# B&R Automation Studio project TD52 (part 135)

#### de_excitCyclic.st
```iecst
(*******************************************************************************
de-excit	 deexcitation generator

This code is confidential and proprietary to the INNIO Company.
It may not be used in any form, or reproduced in any manner,
without the express written permission of the INNIO Company.
Copyright, INNIO Company, 2022

Customized modifications: -
------------------------

History:
-------
V2.12	24.04.2006	LH			copy of gcb
								adapted for de-exitation
		11.11.2006	LH			revised for final release after Para.bMSy test
V3.90.0	09.11.2012	lettenb.	new for modulare software project
		10.05.2013				rU_Gen_Nom --> rU_Gen_Nom[1]
V4.03.0 18.11.2015 	zengerer	BUGFIX Para.rU_Gen_Nom[1] <> 0
V4.07.0 01.02.2019	hohensinner	OUT_SY.bSel_DeExc New interfaces for CU Module (AB Energy like projects and so on), no functionality change in any module done! new INPUT interfaces are not connected! new OUTPUT interfaces are connected!
		17.05.2019	lettenb.	version
V4.09.0	28.11.2019	lettenb.	gen.deexcitation with closing gas valves(before with NOT bN_EngStart), to avoid undefined generator voltage values which may cause unwanted trips of protection relays(ThJ).
V4.10.0	24.11.2019	lettenb.	bMsg2354 added
V4.12.0	14.06.2022	lettenb.	tDemGenExcOff, tGenExcOff added, dead bb synch
		23.11.2022	lettenb.	bDeEx_Dem_x: bOMSS_Man, bOMSS_Aut removed(AA46/wasserer)
								ANW_ENTR: bGnlTrip1 -> bGnlTrip(same condition as for ton_gcb_dmnd_sy)(AA46/wasserer)
V4.13.0	17.08.2023	lettenb.	dead bb synch, bugfixes(BR21/wasserer,schwab,lettenb.)
		20.11.2023	Farre,		added IN_SY.bBypassMCB_SoftStart and soft energisation demand interfaces from CU needed for Microgrid (2023-168)
		29.11.2023	Goenczi,	demand de-exc. from HMI or BUS (e.g. Aggreko)

Instructions for use:
--------------------
Outstandings:
------------
*******************************************************************************)
PROGRAM _CYCLIC

	IF	Para.bSyActive AND Para.bGenDeexit_Enable	THEN

		(*----------------------------------------------------------------------------*)
		(* demand de-excitation *)
		bDeEx_Dem_Man	:=	bSyOMSS_Man
					AND	NOT	gcb.man_off
					AND	   ((gcb.man_on OR ANW_ENTR)
							OR (IN_SY.bOM_Bus				(*	either from HMI or BUS *)
								AND NOT IN_SY.bSetGCB2Open
								AND (IN_SY.bSetGCB2Close OR ANW_ENTR)));

		bDeEx_Dem_Aut	:=	bSyOMSS_Aut
					AND		IN_SY.bEng_Rdy_Aut_Exc;

		IF IN_SY.tDemGenExcOff.Di AND bP_Lo THEN (* dead bus synch *)
			ANW_ENTR	:= (bDeEx_Dem_Man OR bDeEx_Dem_Aut)
						OR (ANW_ENTR AND gcb.on);
		ELSE
			ANW_ENTR	:= (bDeEx_Dem_Man OR bDeEx_Dem_Aut OR IN_SY.bSoftEnergDem)
					AND	    bb_dead
					AND     gcb.eng_oper
					AND NOT gcb.on
					AND 	gcb.rel_trip
					AND 	(IN_SY.bBypassMCB_SoftStart OR (
							NOT		mcb.on
							AND 	mcb.remote
							AND 	mcb.racked_in))
					AND	NOT	bGnlTrip
					AND	NOT	bGen_DeExc_Err;
		END_IF;

		(*----------------------------------------------------------------------------*)
		(* generator de-excited (de-energized) *)
		bGen_DeExc_Rdy	:=	ANW_ENTR AND GEN_OSP;		(* feed-back generator without voltage    *)

		(*----------------------------------------------------------------------------*)
		(* de-excitation finished *)
		tof_T_ENTR(IN:=	ANW_ENTR, PT:= T#5s);

		OUT_SY.bGen_Exc_Off	:=	tof_T_ENTR.Q;

		(*----------------------------------------------------------------------------*)
		(* de-excitation failure *)
		ton_ST_ENTR(IN:= ANW_ENTR AND NOT GEN_OSP, PT:=	T#20s);
		tof_T_ST_ENTR(IN:= ton_ST_ENTR.Q, PT:= T#26s);

		bGen_DeExc_Err	:=	tof_T_ST_ENTR.Q;
		OUT_SY.bGen_DeExc_Rdy := bGen_DeExc_Rdy;
	ELSE
		ANW_ENTR		:= FALSE;
		OUT_SY.bGen_DeExc_Rdy := FALSE;
	END_IF;

	OUT_SY.bSel_DeExc	:=	ANW_ENTR;

		(*----------------------------------------------------------------------------*)
		(* Generator without voltage *)
		IF Para.rU_Gen_Nom[1] <> 0 THEN
			rU_Gen_Norm := IN_SY.tU_Avg[1].Ai / Para.rU_Gen_Nom[1];
		END_IF

		xGR_MIN_GEN_SPG(In:= rU_Gen_Norm, Gw:= Para.rU_Gen_DeEx_LimLo, Hy:= Para.rU_Gen_DeEx_LimLo/5);
		xTON_GEN_OSP(IN:= xGR_MIN_GEN_SPG.Q, PT:= T#1s);

		GEN_OSP := xTON_GEN_OSP.Q;
		OUT_SY.tGenExcOff.Do := GEN_OSP;

		bN_DeExc := IN_SY.rN_EngAct > (Para.rN_EngNom * 0.80);
		bDeEx_EngStop	:=	NOT bN_DeExc 	(* deexcitation at stopped engine, for unitrol reset *)
						AND NOT IN_SY.bGV_On
						AND NOT	IN_SY.bEng_Dem;

		(* Generator de-excitation *)
		bGenDeexitDem := (IN_SY.bMsg1036 OR IN_SY.bMsg1073 OR IN_SY.bMsg1132 OR IN_SY.bMsg1134 OR MM2VIS.bMsg2354 OR IN_SY.bMsg3319 OR ANW_ENTR OR bDeEx_EngStop)
				      AND(NOT IN_SY.tGCB_On.Di OR IN_SY.tDemGenExcOff.Di);
		OUT_SY.tGenDeexitDem.Do := bGenDeexitDem;

		(*----------------------------------------------------------------------------*)

END_PROGRAM
```

#### de_excit.var
```iecst
VAR
	bDeEx_Dem_Man : BOOL;
	bDeEx_Dem_Aut : BOOL;
	tof_T_ENTR : TOF;
	ton_ST_ENTR : TON;
	tof_T_ST_ENTR : TOF;
	xGR_MIN_GEN_SPG : GR_MINR;
	xTON_GEN_OSP : TON;
	bDeEx_EngStop : BOOL;
	bN_DeExc : BOOL;
END_VAR
```

### Program Logical/Synchronization/blackstart (IEC, version 4.13.0) - blackstart procedure

#### blackstartCyclic.st
```iecst
(*******************************************************************************
blackstart		blackout start

This code is confidential and proprietary to the INNIO Company.
It may not be used in any form, or reproduced in any manner,
without the express written permission of the INNIO Company.
Copyright, INNIO Company, 2022

Customized modifications: -
------------------------

History:
-------
V2.12	24.04.2006	LH			adapted for esy new
		02.10.2006	LH			modification of anti-detonation logic
		16.10.2006	LH			for execution load shedding:
								dmnd_load_shedd --> dmnd_black_start
		31.10.2006	LH			adaption of island release coming from Para.bMSy
		11.11.2006	LH			revised after Para.bMSy test
		20.11.2006	LH			revised for final release esy new
V2.20	27.04.2007	LH			update according to last changes mcb(s)
V2.20.1	08.08.2007	LH			termination of island power monitoring
V2.30	18.01.2008	LH			adapted for test-bench run
V3.99.0	04.03.2013	lettenb.	adapted for pilot engine 612, update anti detonation logic
		04.07.2013				IN_SY.tP_MnsImp_Act --> IN_SY.rP_MainsImport from MM_CU
V4.00.0 12.06.2014	lettenb.	test bTestBenchModeIsland
V4.03.0 18.11.2015  zengerer	BUGFIX NULLDIVISIONEN AND IN_SY.rP_Nom > 0
		11.04.2016	lettenb.	ton_dmnd_bs_over.Q -> dmnd_bs_over, bugfix
V4.12.0 29.06.2022	lettenb.	dead bb synch
V4.13.0 23.05.2023	Goenczi		code array view, interfaces from CU

Instructions for use:
--------------------

Outstandings:
------------
monitoring pmin in island operation ? (in v3.40 not active)
*******************************************************************************)
FUNCTION AND_Array
	memcpy(ADR(Arrayx),Adress,MIN(40,Size) + 1);
	AND_Array	:=	 TRUE;
	FOR i:= 0 TO MIN(40,Size) DO
		AND_Array	:=	AND_Array AND Arrayx[i];
	END_FOR
END_FUNCTION

FUNCTION OR_Array
	memcpy(ADR(Arrayx),Adress,MIN(40,Size) + 1);
	OR_Array	:=	 FALSE;
	FOR i:= 0 TO MIN(40,Size) DO
		OR_Array	:=	OR_Array OR Arrayx[i];
	END_FOR
END_FUNCTION

PROGRAM _CYCLIC

	IF	Para.bSyActive	THEN
		(*----------------------------------------------------------------------------*)
		(* general release island operation *)
		xTON_Sys_Run(IN:= IN_SY.tPB2MM.bSys_Run, PT:= T#10s);

		bIsl_mode[0]	:=	gcb.rel_island AND gcb.eng_oper AND gcb.other_gen_parallel AND	NOT	tof_mns_connection.Q;
		bIsl_mode[1]	:=	gcb.rel_island AND NOT OUT_SY.bSmoothDischarge;
		bIsl_mode[2]	:=	OUT_SY.bOnly_Island;

		bIsland_mode	:=	OR_Array(ADR(bIsl_mode),2);

		bRel_Isl[0]	:=	Para.bIslandOp_Enable OR Para.bOnlyIsland_Enable OR Para.bMSy OR Para.bMCB_Ctr_Cust	OR OUT_SY.bTestBenchModeIsland;
		bRel_Isl[1]	:=	IN_SY.tRel_I.Di;	(* release island extern (OUT_SY.bRel_Island)   *)
		bRel_Isl[2]	:=	xTON_Sys_Run.Q;
		bRel_Isl[3]	:=	bIsland_mode;
		bRel_Isl[4]	:=	IN_SY.bRel_I_Bus;	(*release island via Bus*)
		bRel_Isl[5]	:=	IN_SY.bCust_Rel_I;	(*custom release from CU*)

		bRelease_Island	:=	AND_Array(ADR(bRel_Isl),5);

		(* release island operation busbar: false = mains-cut-off with gcb *)
		bRel_Isl_BB[0]	:=	gcb.on AND bDem_Island AND NOT mcb.on;
		bRel_Isl_BB[1]	:=	gcb.on AND NOT sel_gcb_mains_cut_off AND NOT MM2VIS.bMsg3412;
		bRel_Isl_BB[2]	:=	other_gcb_on;
		bRel_Isl_BB[3]	:=	dmnd_black_start;
		bRel_Isl_BB[4]	:=	IN_SY.bCust_RelI_BB; 	(*new Aggreko release from CU*)
		bRel_Isl_BB[5]	:=	FALSE;

		bRelease_Isl_BB	:=	OR_Array(ADR(bRel_Isl_BB),5);

		bRel_VKE10[0]	:=	bRelease_Isl_BB;
		bRel_VKE10[1]	:=	bRelease_Island;
		bRel_VKE10[2]	:=	NOT	mcb.alm_psf OR	OUT_SY.bTestBenchModeIsland;
		bRel_VKE10[3]	:=	NOT	mcb.alm_opf;
		bRel_VKE10[4]	:=	NOT	any_gcb_opf_bb;

		bRelease_VKE10	:=	AND_Array(ADR(bRel_VKE10),4);

		(* demand island operation (INSEL) *)
		bDem_Isl[0]	:=	bRelease_VKE10;
		bDem_Isl[1]	:=	rel_i_adl OR NOT Para.bADL_Enable; (* release from anti-detonation logic *)

		bDem_Island	:=	AND_Array(ADR(bDem_Isl),1);

		(*----------------------------------------------------------------------------*)
		(* release black-out start *)
		rel_black_start	:= (Para.bBS_Enable OR Para.bOnlyIsland_Enable OR Para.bMSy	OR OUT_SY.bTestBenchModeIsland)
					AND		IN_SY.tRel_BS.Di;			(* release black-out extern (BL_OUT) *)

		(*----------------------------------------------------------------------------*)
		(* demand black-out start (BLOUT) *)
		black_status_bb := (all_gcb_off_bb OR IN_SY.tDemGenExcOff.Di)
					AND		mcb.off;

		(*----------------------------------------------------------------------------*)
		IF NOT Para.bMCB_ReSw2Mns_Enable THEN
			dmnd_black_start :=	bRelease_Island					(* BLOUT *)
						AND		rel_black_start
						AND	   (bSyOMSS_Man OR	NOT	Para.bBS_OnlyMan)
						AND	   (bOMSS_Man   OR	NOT	Para.bBS_OnlyMan)
						AND(NOT bMainsReturn					    OR black_status_bb)
						AND	   (mcb.off     OR  NOT MM2VIS.bMsg3412 OR black_status_bb)
						AND   	mcb.remote
						AND(NOT	mcb.alarm   OR	    OUT_SY.bTestBenchModeIsland)
						AND NOT any_gcb_alarm_bb
						AND NOT	dmnd_bs_over;

		ELSIF Para.bMCB_ReSw2Mns_Enable THEN
			dmnd_black_start :=	bRelease_Island					(* BLOUT *)
						AND		rel_black_start
						AND	   (bSyOMSS_Man OR	NOT	Para.bBS_OnlyMan)
						AND	   (bOMSS_Man   OR	NOT	Para.bBS_OnlyMan)
						AND	NOT bMainsReturn
						AND	   (mcb.off     OR  NOT MM2VIS.bMsg3412)
						AND   	mcb.remote
						AND(NOT	mcb.alarm   OR	    OUT_SY.bTestBenchModeIsland)
						AND NOT any_gcb_alarm_bb
						AND NOT	dmnd_bs_over;
		END_IF;

		(*----------------------------------------------------------------------------*)
		(* black-out start procedure finished *)
		dmnd_bs_over	:= (dmnd_black_start OR	dmnd_bs_over)
					AND		gcb.eng_oper
					AND		gcb.on;

		(*----------------------------------------------------------------------------*)
		(* demand load shedding *)
		dmnd_load_shedd	:=	black_status_bb
					AND		bRelease_Island
					AND		rel_black_start
					AND		dmnd_black_start;

		(* load shedding ok *)
		ton_ls_ok(IN:= dmnd_load_shedd AND IN_SY.tRel_LS.Di, PT:= T#5s);

		rel_load_shedd	:=	ton_ls_ok.Q;		(* load shedding is done (LAST_AB) *)

		(******************************************************************************)
		(* anti detonation logic *)
		(*----------------------------------------------------------------------------*)
		tof_mns_connection(IN:= mcb.on, PT:= T#5s);	(* mains connected to busbar	 *)
		ton_gcb_on        (IN:=	gcb.on, PT:= T#5s);	(* generator connected to busbar *)

		(*----------------------------------------------------------------------------*)
		IN_SY.rP_Nom;						(* engine nominal generator power [kW] *)
		IN_SY.rP_Act_Norm_Filt;				(* engine actual  generator power [kW] *)

		rPchange_max	:=	40.0;			(* maximum allowed loss of gen. power *)
		rPgen_min		:=	15.0;			(* minimum required island power      *)

		(*----------------------------------------------------------------------------*)
		(* generator power supplied to busbar *)
		IF gcb.on THEN	rP_Gen_Act_Norm := IN_SY.rP_Act_Norm_Filt;
		ELSE			rP_Gen_Act_Norm := 0.0;
		END_IF;

		(* mains power to busbar in % Pnom engine *)
		IF mcb.on AND IN_SY.rP_Nom > 0  THEN	rP_Mns_Act_Norm := IN_SY.rP_MainsImport / IN_SY.rP_Nom;
		ELSE			rP_Mns_Act_Norm := 0.0;
		END_IF;

		(* consumer load on busbar *)
		rP_Csm_Act_Norm := rP_Gen_Act_Norm + rP_Mns_Act_Norm;

		(*----------------------------------------------------------------------------*)
		(* release for island operation *)
		IF (Para.bMSy AND mcb.on AND bRelease_VKE10) OR NOT mcb.on THEN
			rel_i_adl		:=	TRUE;
		ELSIF NOT VKE41 AND mcb.on	THEN
			rel_i_adl		:=	TRUE;					(* cond. to change into island are ok *)
		ELSE
			rel_i_adl		:=	FALSE;					(* change into island is not allowed  *)
		END_IF;

		(*----------------------------------------------------------------------------*)
		(* monitoring change of generator power in case of opening mcb *)
		VKE40			:=	VKE41						(* maintained lock command            *)
					AND	NOT	gcb.on
					AND		gcb.eng_run;

		VKE41			:=	VKE40						(* --> lock module after opening xcb  *)
					OR	   (rPchange > rPchange_max);	(* because of too much loss of power  *)

		(* --> no load expected because:  *)
		bPcalc		:=		mcb.on								(* - no connection to mains          *)
					AND		bRelease_VKE10						(* - no island operation selected    *)
					AND		(IN_SY.rP_MainsImport <> -999999.0)	(* - no mains power signal, value if signal not connected = -999999 from MM_CU *)
					AND		other_gcb_off;						(* - Pcsm calculation  not possible	*)

		IF	bPcalc	THEN
			rP_I_Act_Norm_Expected := rP_Csm_Act_Norm;	(* gen.load will be consumer load   *)
		ELSE
			rP_I_Act_Norm_Expected := 0;				(* no load expected at opening xcb    *)
		END_IF;

		(* change of gen. power at opening xcb = generator power supplied to busbar - expect.load in case of opening mcb*)
		rPchange	:=	IN_SY.rP_Act_Norm_Filt - rP_I_Act_Norm_Expected;

		(*----------------------------------------------------------------------------*)

	END_IF;

END_PROGRAM
```

#### blackstartInit.st
```iecst
PROGRAM _INIT
	(* init program *)

	rPel_csm_old	:=	10000.0;

END_PROGRAM
```

#### blackstart.fun
```iecst
(********************************************************************
 * COPYRIGHT -- INNIO Company
 ********************************************************************
 * Package: blackstart
 * File: blackstart.fun
 * Author: 212426533
 * Created: November 29, 2023
 *******************************************************************)

FUNCTION AND_Array : BOOL
	VAR_INPUT
		Adress : UDINT;
		Size : USINT;
	END_VAR
	VAR
		i : USINT;
		Arrayx : ARRAY[0..40] OF BOOL;
	END_VAR
END_FUNCTION

FUNCTION OR_Array : BOOL
	VAR_INPUT
		Adress : UDINT;
		Size : USINT;
	END_VAR
	VAR
		i : USINT;
		Arrayx : ARRAY[0..40] OF BOOL;
	END_VAR
END_FUNCTION
```

#### blackstart.var
```iecst
VAR
	rPchange : REAL;
	rPchange_max : REAL;
	rPel_csm_old : REAL;
	rPgen_min : REAL;
	rP_Gen_Act_Norm : REAL;
	rP_Mns_Act_Norm : REAL;
	rP_Csm_Act_Norm : REAL := 0.0;
	tof_mns_connection : TOF;
	ton_gcb_on : TON;
	ton_ls_ok : TON;
	black_status_bb : BOOL;
	xTON_Sys_Run : TON;
	dmnd_bs_over : BOOL;
	bRelease_VKE10 : BOOL; (* release island operation busbar: false = mains-cut-off with gcb *)
	VKE40 : BOOL;
	VKE41 : BOOL;
	bPcalc : BOOL;
	dmnd_load_shedd : BOOL; (*Demand load shed*)
	rP_I_Act_Norm_Expected : REAL;
	bIsl_mode : ARRAY[0..2] OF BOOL := [3(0)];
	bIsland_mode : BOOL := 0;
	bRel_Isl : ARRAY[0..5] OF BOOL := [6(0)];
	bRel_Isl_BB : ARRAY[0..5] OF BOOL := [6(0)]; (* release island operation busbar condition OR array: false = mains-cut-off with gcb *)
	bRelease_Isl_BB : BOOL := 0; (* release island operation busbar part1 *)
	bDem_Isl : ARRAY[0..1] OF BOOL := [2(0)]; (* demand island operation (INSEL) condition array*)
	bRel_VKE10 : ARRAY[0..4] OF BOOL := [5(0)]; (* release island operation busbar condition AND array: false = mains-cut-off with gcb *)
END_VAR
```

### Program Logical/Synchronization/sy_out (IEC, version 4.13.0) - out signals handling

#### sy_outCyclic.st
```iecst
(*******************************************************************************
sy_out		control outputs

This code is confidential and proprietary to the INNIO Company.
It may not be used in any form, or reproduced in any manner,
without the express written permission of the INNIO Company.
Copyright, INNIO Company, 2022

Customized modifications: -
------------------------

History:
-------
V2.12	24.04.2006	LH			gcb1 imported from MSY
								gcb1 --> sy_out
								adapted for esy new
		31.10.2006	LH			insert release gcb from Para.bMSy
		11.11.2006	LH			revised after Para.bMSy test
		20.11.2006	LH			revised for final release esy new
V2.20	07.02.2007	LH			new: lock command for customer mcb
		19.02.2007	LH			adapted for X20-system
								advanced software documentation
		04.04.2007	LH			correction of OUT_SY.bRel_IslandAfMITime in case of mcb controlled by customer
V2.201	22.05.2007	TW			change MMU variables to array (ex task: DO)
V2.30	16.01.2008	LH			building OUT_SY.bRel_IslandAfMITime to prevent engine shutdown
								during waiting time for island demand
		18.01.2008	LH			adapted for test-bench run
V2.30	22.02.2008	LH			change output gcb opening failure (ex task: DO)
		26.02.2008	LH			connect gcb position sig. fail. to engine control
		05.03.2008	LH			change gcb position sig. fail. to engine control
								to undelayed tripping
		28.03.2008	LH			connect gcb closing failure to engine control
V2.34.0	19.12.2008	lettenb.	OUT_SY.bRelEngOpFromSY: gcb.mdl removed
V2.60.0	13.08.2009	lettenb.	gcb_opf_delay for opening mcb with delay added (ex task: DO)
V2.60.0	08.10.2009	lettenb.	ton_dmnd_synchline added (delay for activating synch.device
 								after switching on the voltage signals to the synch.device.
								MMUsynch needs some time until frequence measuring is ok)
V3.20.0	01.07.2010	lettenb.	BR9_B added
		13.01.2011	lettenb.	Para.bEngOpAfterMIF_Enable added
V3.20.0	04.11.2010	lettenb.	bSyncSlipMode[2], bMMU2syMCB added for synchr.mcb with MMU2 (ex task: DO)
V3.30.0 02.02.2012	lettenb.	OUT_SY.bEng_Dem_EPS_Sy: Para.bIslandOp_Enable	added(to avoid message 'demand emerg.operation'
								in case of mains break down and no island operation is selected)
V3.90.0	13.11.2012	lettenb.	parts from pb17_en included
V3.99.0 26.02.2013	lettenb.	task DO included, iEngNr added
V3.99.1	25.03.2013	Denk		bRelSyFromCU changed to bRelSy_Customized
		27.06.2013	lettenb.	bRelEng4OnlyI_Op: brackets added, bugfix
V4.00.0 11.06.2014	lettenb.	bRelEng4I_Op: logic, ton_BLO_AES.PT case iEngNr, bugfix
		16.06.2014	lettenb.	OUT_SY.bRelEngOpFromSy: IN_SY.tMCB_Rel_Sync_SOn.Do ERDF lockout added (grid)
V4.04.0 31.10.2016				ton_esl.IN: ... AND FALSE) (* FALSE=econ_lock; added, acc.a_V3.59, wasserer/rosenheim)
        05.12.2016				OUT_SY.tRdy_MSy.Do,OUT_SY.tEng_Run_Sy.Do,OUT_SY.tEng_Dem.Do always active for GSY
		01.10.2020	lettenb.	OUT_SY.bMCB_DemSy, mcb controlled by customer, bugfix(heim, Referenzanlage AB85), bu
V4.10.0 15.12.2020	lettenb.	BR6 release island after MIF: bRel_IslandAfMITime in case of Para.bP_LoadReject_Active AND IN_SY.bType6_Update_Rel
V4.12.0 24.11.2020	lettenb.	WaitingTime_CloseGCB2DeadBB_too_long issue#911
								xTOF_RelEng4I_Op added, avoid loss of RelEng4I_Op for 1 cycle at OMSS change to OFF in island, issue#957
V4.13.0	17.08.2023	lettenb.	dead bb synch, bugfixes(BR21/wasserer,schwab,lettenb.)
		19.07.2023	Goenczi		Added Para.bSel_Customer to bRelEng4I_Op to bypass Dem_Island for Aggreko
								bEng_Dem_EPS_Sy condition from CU module added

Instructions FOR use:
--------------------
						variante:	ESy		+Msy	+CCB	noSy	GSy		AB_Sy
	immer	A_USP
			DO_ENG_D
			DO_PUL_MNS_OK
			DO_GCB_REL
			DO_GCB_RSP
			DO_GCB_OPF
			DO_GCB_CON
			DO_GCB_COF
			DO_GCB_RT

	msy		DO_GCB_ESL
			DO_GCB_EDC
			DO_RDY_MSY
			DO_ENG_RUN		OUT_SY.tEng_Run.Do;

	mcb		DO_MCB_RSP
			DO_MCB_DVS
			DO_MCB_RT
			DO_MCB_CON
			DO_MCB_COF

	AB		A_SYANW
			A_RSYANW

	indon.	DO_DMND_LS

Outstandings:
------------
define variations by parameter-settings
*******************************************************************************)
PROGRAM _CYCLIC

	IF	Para.bSyActive	THEN
		(*----------------------------------------------------------------------------*)
		(* demand synchline *)			(* OUT_SY.bDSyLine *)
		ton_dmnd_synchline(IN:= (gcb.dmnd_sy OR mcb.dmnd_sy) AND NOT pulse_sy_line, PT:= T#2s);

		dmnd_synchline := ton_dmnd_synchline.Q;

		(*----------------------------------------------------------------------------*)
		(* ESy demand lock all other cb's for closing gcb to dead busbar *)		(* BLO_AES) *)
		ton_BLO_AES.IN	:= (ton_gcb_dmnd_sy.IN	OR ton_gcb_dmnd_sy.Q)
					AND(    bb_dead OR(IN_SY.tDemGenExcOff.Di AND NOT bb_alive))(* dead busbar (OUT_SY.bBB_dead) *)
					AND(NOT	MM2VIS.bMsg1216	OR	OUT_SY.bTestBenchModeIsland)	(* no busbar voltage sensor failure *)
					AND(NOT any_gcb_on_bb   OR  IN_SY.tDemGenExcOff.Di)			(* all gcb open - busbar *)
					AND	NOT any_gcb_psf_bb										(* no other gcb with position failure *)
					AND NOT any_gcb_opf_bb										(* no other gcb with opening failure *)
					AND NOT mcb.on												(* all mcb open *)
					AND(NOT mcb.alm_psf		OR	OUT_SY.bTestBenchModeIsland)	(* no mains cb with position failure *)
					AND		IN_SY.tPB2MM.bSys_Run;								(* CPU is alive *)

		IF Para.bMSy THEN
			ton_BLO_AES.PT	:=	T#1s;		(* gcb close2deadBB interlock is done MSy *)
		ELSE
			CASE iEngNr OF
			1:	ton_BLO_AES.PT	:=	T#1s;	(* engine 1 *)
			2:	ton_BLO_AES.PT	:=	T#2s;
			3:	ton_BLO_AES.PT	:=	T#3s;
			4:	ton_BLO_AES.PT	:=	T#4s;
			5:	ton_BLO_AES.PT	:=	T#5s;
			6:	ton_BLO_AES.PT	:=	T#6s;
			7:	ton_BLO_AES.PT	:=	T#7s;
			8:	ton_BLO_AES.PT	:=	T#8s;
			9:	ton_BLO_AES.PT	:=	T#9s;
			10:	ton_BLO_AES.PT	:=	T#10s;
			11:	ton_BLO_AES.PT	:=	T#11s;
			12:	ton_BLO_AES.PT	:=	T#12s;
			13:	ton_BLO_AES.PT	:=	T#13s;
			14:	ton_BLO_AES.PT	:=	T#14s;
			15:	ton_BLO_AES.PT	:=	T#15s;
			16:	ton_BLO_AES.PT	:=	T#16s;
			ELSE
				ton_BLO_AES.PT	:=	T#17s;
			END_CASE;
		END_IF;
		ton_BLO_AES();

		gcb.edc		:=	ton_BLO_AES.Q									(* demand closing gcb to dead busbar *)
					OR	mcb_man_on2dead_bb								(* manual closing mcb1 to dead busbar *)
					OR	mcb_aut_on2dead_bb;								(* automatic closing mcb1 to dead busbar *)

		(* ESY demand lock customer mcb while running island operation *)
		BLOCK_NS		:=	ton_BLO_AES.Q								(* demand closing gcb to dead busbar *)
					OR(			BLOCK_NS
						AND		any_gcb_on_bb							(* lock customer mcb will last until *)
						AND	NOT	mcb.dmnd_sy);							(* resynchronizing is initiated *)

		(* release closing cb to dead busbar to MSY/external unit (AES_FRG) *)
		ton_esl.IN		:= (bb_dead AND NOT	ton_gcb_dmnd_sy.IN AND IN_SY.tPB2MM.bSys_Run AND NOT gcb.release AND FALSE) (* FALSE= ex.econ_lock;	interlock cb's only with 1 signal ? *)
					OR	   (any_gcb_edc_bb	                   AND IN_SY.tPB2MM.bSys_Run AND NOT gcb.release)			(* demand closing ext. cb to dead busbar (ANF_BLO) *)
					OR	   (gcb.mdl                            AND IN_SY.tPB2MM.bSys_Run AND NOT gcb.release);			(* demand lock from MSy *)
		ton_esl(PT:= T#1s);												(* engine (gcb) status locked -> release gcb (FG_GS) *)

		gcb.esl		:=	ton_esl.Q;										(* release closing ext. cb to dead busbar (AES_FRG) *)

		(*----------------------------------------------------------------------------*)
		(* demand emergency operation (OUT_SY.bEng_Dem_EPS_Sy) *)
		OUT_SY.bEng_Dem_EPS_Sy	:= ((Para.bIslandOp_Enable OR Para.bOnlyIsland_Enable OR Para.bMSy OR Para.bMCB_Ctr_Cust)
							AND(NOT	mains.ok OR	NOT	mcb.on)
							AND IN_SY.bCust_Dem_EPS_Sy);

		(*----------------------------------------------------------------------------*)
		(* release engine operation from ESY (OUT_SY.bRelEngOpFromSY) *)
		bRelEng4NP_Op	:= (mains.ok OR gcb.eng_oper)					(* release for parallel operation *) (* mehrfachverwendung *)
					AND		mcb.on										(* mcb closed (NS(1)_EIN) *)
					AND		bMainsReturn								(* mains return (OUT_SY.bMainsReturn) *)
					AND	NOT	MM2VIS.bMsg3412;							(* mains monitoring device failure *)

		(*----------------------------------------------------------------------------*)
		(* hold release engine for island op. after mi-filter time *)
		xTOF_Rel_IslandAfMITime(IN:= mains.ok, PT:= T#60s);

		IF 			NOT	gcb.eng_oper									(* no engine operation (IN_SY.tEng_Run.Do) *)
				OR	NOT	Para.bMIF_Enable
				OR		Para.bBS_OnlyMan
				OR	NOT	Para.bEngOpAfterMIF_Enable
				OR	   (xEngType.Type6 AND (NOT Para.bP_LoadReject_Active OR NOT IN_SY.bType6_Update_Rel))
				OR		xEngType.Type9
		THEN
			xTOF_Rel_IslandAfMITime(IN:= FALSE, PT:= T#0s); 			(* reset bridging *)
		END_IF;

		OUT_SY.bRel_IslandAfMITime	:=	xTOF_Rel_IslandAfMITime.Q;		(* prevention of engine shutdown (M_BLOCK) *)
		(*----------------------------------------------------------------------------*)

		(* hold release engine for island op. for reswitch to mains *)
		xTOF_Rel_Island4Resw2Mns(IN:= gcb.on, PT:= T#60s);

		IF		NOT	gcb.eng_oper										(* no engine operation (IN_SY.tEng_Run.Do) *)
			OR	NOT	Para.bMCB_ReSw2Mns_Enable
			OR		Para.bBS_OnlyMan
			OR	   (xEngType.Type6 AND (NOT Para.bP_LoadReject_Active OR NOT IN_SY.bType6_Update_Rel))
			OR		xEngType.Type9
		THEN
			xTOF_Rel_Island4Resw2Mns(IN:= FALSE, PT:= T#0s);			(* reset bridging *)
		END_IF;

		bRel_Island4Resw2Mns := xTOF_Rel_Island4Resw2Mns.Q;

		(*----------------------------------------------------------------------------*)
		xTOF_RelEng4I_Op(IN	:= (Para.bIslandOp_Enable OR Para.bMSy OR Para.bMCB_Ctr_Cust OR OUT_SY.bTestBenchModeIsland)
						AND	   (rel_i_adl OR NOT Para.bADL_Enable)
						AND	   (OUT_SY.bRel_IslandAfMITime OR bRel_Island4Resw2Mns OR bDem_Island OR gcb.rel_trip OR Para.iSel_Customer = 2), PT:= T#200ms);
		bRelEng4I_Op	:= xTOF_RelEng4I_Op.Q;

		bRelEng4OnlyI_Op:=	OUT_SY.bOnly_Island
					AND		mcb.off
					AND	NOT	mcb.on
					AND	  ((OUT_SY.bRelEngOpFromSy AND(gcb.eng_oper OR gcb.eng_demanded)) OR NOT gcb.eng_run);

		bRelEng4Op		:=	mcb.remote
					AND		mcb.racked_in
					AND		gcb.racked_in
					AND  (((bRelEng4NP_Op OR bRelEng4I_Op) AND NOT OUT_SY.bOnly_Island) OR bRelEng4OnlyI_Op);	(* release for island/parallel operation *)

		OUT_SY.bRelEngOpFromSy := 	IN_SY.tLineCB_On.Di
								AND IN_SY.bRelSy_Customized				(* from MM_CU *)
								AND bRelEng4Op
								AND IN_SY.tMCB_Rel_Sync_SOn.Do;			(* ERDF lockout *)
	ELSE

		OUT_SY.bRelEngOpFromSy := 	IN_SY.tLineCB_On.Di
								AND IN_SY.bRelSy_Customized 			(* from MM_CU *)
								AND IN_SY.tRelEngOpFromGSy.Di
								AND IN_SY.tMCB_Rel_Sync_SOn.Do;			(* ERDF lockout *)
	END_IF;

	(*-----------------------------------------------------------------------------*)
	(* diagnostics *)
	bRelEng4NP_Op;				(* release engine for net parallel *)
	bRelEng4I_Op;				(* release engine for island(emergency op.)*)
	bRelEng4OnlyI_Op;			(* release engine for only island *)
	OUT_SY.bRelEngOpFromSy;		(* release engine for operation from sy *)
	(*-----------------------------------------------------------------------------*)

	(*-----------------------------------------------------------------------------*)
	(* switch standard-inputs esy to required inputs engine control *)
		OUT_SY.bSynchDem		:=		IN_SY.tGCB_DSY.Di;				(* demand synchline *)

		(* general -------------------------------------------------------------------*)
		OUT_SY.tRdy_MSy.Do		:=		IN_SY.bEng_Rdy_Aut_Exc;			(* engine ready    for MSY/GSY *)
		OUT_SY.tEng_Run_Sy.Do	:=		bN_EngStart;					(* engine rotating for MSY/GSY *)
		OUT_SY.tEng_Dem.Do		:=		IN_SY.bEng_RPSDem;				(* engine demanded for MSY/GSY *)
		OUT_SY.tOMSS_Man.Do		:=		bOMSS_Man;						(* oper.mode man.  for     GSY *)
		OUT_SY.tOMSS_Aut.Do		:=		bOMSS_Aut;						(* oper.mode aut.  for     GSY *)

	IF	Para.bSyActive	THEN
		OUT_SY.tDemandBB.Do		:=		gcb.dmnd_sy;					(* demand busbar *)

		OUT_SY.tGCB_ESL.Do		:=		gcb.esl;						(* ESY status gcb locked *)
		OUT_SY.tGCB_EDC.Do		:=		gcb.edc;						(* ESY demand lock all other cb's connected to dead busbar *)
		OUT_SY.tLock_C_MCB.Do	:=		BLOCK_NS;						(* demand lock customer mcb while running island operation *)
		OUT_SY.tGCB_OpF.Do		:=		gcb_opf_delay;					(* alarm gcb opening failure *)

		(* generator circuit breaker -------------------------------------------------*)
		OUT_SY.tGCB_Rel.Do		:=		gcb.release;					(* release closing gcb *)
		OUT_SY.tGCB_RSP.Do		:=		gcb.rel_sy_puls;				(* release sy pulse gcb *)
		OUT_SY.tGCB_COn.Do		:=		gcb.command_on;					(* command gcb on *) (* Do = true  = command ON  *)
		OUT_SY.tGCB_COf.Do		:=	NOT gcb.command_off;				(* command gcb off *)(* Do = false = command OFF, closed circuit principle *)
		OUT_SY.tGCB_RT.Do		:=		gcb.rel_trip;					(* release trip gcb *)
		OUT_SY.tGCB_DVS.Do		:=		gcb.dmnd_sy;					(* demand synchronization gcb - select voltage *)

		(* mains circuit breaker -----------------------------------------------------*)
		OUT_SY.tMCB_RSP.Do		:=	NOT Para.bMSy AND mcb.rel_sy_puls;	(* release sy pulse mcb1 *)
		OUT_SY.tMCB_COn.Do		:=	NOT Para.bMSy AND mcb.command_on;	(* command mcb1 on *)
		OUT_SY.tMCB_COf.Do		:=	NOT Para.bMSy AND mcb.command_off;	(* command mcb1 off *)
		OUT_SY.tMCB_RT.Do		:=	NOT Para.bMSy AND mcb.rel_trip;		(* release trip mcb1 *)
		OUT_SY.tMCB_DVS.Do		:=	NOT Para.bMSy AND mcb.dmnd_sy;		(* demand synchronization mcb1 - select voltage *)

		(* switch standard-outputs esy to standard-inputs engine control -------------*)
		OUT_SY.bMsg1217			:=		gcb.alm_psf;					(* alarm gcb position signal failure *)
		OUT_SY.bMsg1218			:=		gcb.alm_opf;					(* alarm gcb opening failure *)
		OUT_SY.bMsg1219			:=		gcb.alm_cf;						(* alarm gcb closing failure *)
		bGCB_GnlWarning			:=		gcb.alarm;						(* gcb general warning *)
		OUT_SY.bMsg1209			:=		mcb.alm_psf;					(* alarm mcb position signal failure *)
		bMCB_GnlWarning			:=		mcb.alarm;						(* mcb general warning *)

		OUT_SY.bGCB_DemSy		:=		gcb.dmnd_sy;					(* demand synchronization gcb for main loop display *)
		OUT_SY.bMCB_DemSy		:=		mcb.dmnd_sy AND Para.bMCB_Enable;(* demand synchronization mcb for main loop display *)
		OUT_SY.bDSyLine			:=		dmnd_synchline;					(* ESY demand synchline for synchronizing gcb *)
		OUT_SY.bMnsOk			:=		IN_SY.tMnsOk.Di;				(* mains ok       for W1175 *)
		OUT_SY.bMainsReturn		:=		bMainsReturn;					(* mains return   for W1175 and block engine *)
		OUT_SY.bBB_dead			:=		bb_dead;						(* busbar dead for main loop display and B2139/B3265 *)
		OUT_SY.bRel_Island		:=		bRelease_Island;				(* release island for W1175 and block engine *)
		BLOUT					:=		dmnd_black_start;				(* demand black-out start for demand load shedding *)
		OUT_SY.bOtherGenParallel:=		OUT_SY.bOtherGenParallel;		(* other engine parallel for demand emergency op. *)

		(* switch standard-outputs esy new to standard-inputs MMU/Sync ---------------*)
		OUT_SY.bSyncSlipMode[1] :=	   (OUT_SY.bMCB_DemSy	AND NOT Para.bMCB_SyMMD2)	(* synchronization with slip mode *)
									OR (OUT_SY.bGCB_DemSy	AND	NOT	bb_dead);
		OUT_SY.bSyncSlipMode[2] :=  	OUT_SY.bMCB_DemSy	AND 	Para.bMCB_SyMMD2;	(* synchronization with slip mode *)

		(*----------------------------------------------------------------------------*)
		(* synchronizing device on *)			(* SYG_EIN *)
		OUT_SY.bGen_SyD_Dem 	:= (gcb.dmnd_sy OR mcb.dmnd_sy) AND	bb_alive;

		(* release synchronizing pulse *)		(* FG_SYIMP *)
		ton_dmnd_sy_device(IN:= OUT_SY.bGen_SyD_Dem, PT:= T#2s);
		rel_sy_puls				:=	ton_dmnd_sy_device.Q;

		(*----------------------------------------------------------------------------*)
	END_IF;

END_PROGRAM
```

#### sy_out.var
```iecst
VAR
	ton_BLO_AES : TON;
	ton_esl : TON;
	xTOF_Rel_IslandAfMITime : TOF;
	xTOF_Rel_Island4Resw2Mns : TOF;
	ton_dmnd_synchline : TON;
	bRel_Island4Resw2Mns : BOOL;
	bRelEng4NP_Op : BOOL; (* release engine for net parallel operation*)
	bRelEng4I_Op : BOOL; (* release engine for island operation*)
	bRelEng4OnlyI_Op : BOOL; (* release engine for only island operation*)
	bRelEng4Op : BOOL;
	ton_dmnd_sy_device	:TON;
	xTOF_RelEng4I_Op : TOF;
END_VAR
```

### Program Logical/Synchronization/vis_SY (IEC, version 4.13.0) - visualization

#### vis_SYCyclic.st
```iecst
(*******************************************************************************
vis_SY			visualization

This code is confidential and proprietary to the INNIO Company.
It may not be used in any form, or reproduced in any manner,
without the express written permission of the INNIO Company.
Copyright, INNIO Company, 2022

Customized modifications: -
------------------------

History:
-------
V3.90.0	17.10.2012	lettenb.	new
V3.99.0	04.03.2013	lettenb.	new version
V4.07.0	11.10.2018	lettenb.	DI/DO dataitems for diagnosis added
 		25.04.2019	lettenb.	dataitem changed IN_SY.tGCB_DVM.Di, bugfix
		01.10.2020	lettenb.	MM2VIS.bDSyMCB, mcb controlled by customer, bugfix(heim, Referenzanlage AB85), bu
V4.12.0	14.09.2022	lettenb.	MM2VIS.bDemGenExcOff, MM2VIS.bGenExcOff added, dead bb synch
V4.13.0	29.11.2023	Goenczi		bGCB_OGP_Bus other genset paralell bit via bus

Instructions for use:
--------------------
Outstandings:
------------
*******************************************************************************)
PROGRAM _CYCLIC

	MM2VIS.bMnsOk			:=		OUT_SY.bMnsOk;		(* mains ok *)
	MM2VIS.bNotMainsReturn	:=	NOT	bMainsReturn;		(* not mains return *)

	MM2VIS.bGCB_On			:=		IN_SY.tGCB_On.Di;	(* gcb closed for report time measuring *)
	MM2VIS.bGCB_GnlWarning	:=		bGCB_GnlWarning;	(* gcb general failure *)
	MM2VIS.bDSyGCB			:=		gcb.dmnd_sy;		(* gcb demand synchronization *)

	MM2VIS.bMCB_On			:=		OUT_SY.bMCB_On;		(* mcb closed for report time measuring *)
	MM2VIS.bMCB_GnlWarning	:=		bMCB_GnlWarning;	(* mcb general failure *)
	MM2VIS.bDSyMCB			:=		mcb.dmnd_sy AND Para.bMCB_Enable;	(* mcb demand synchronization *)

	MM2VIS.bEngDemIsland 	:=		IN_SY.tEngDemIsland.Di;	(* DI engine demand for island operation *)
	MM2VIS.bOnly_Island		:=		IN_SY.tOnly_Island.Di;	(* DI only island operation *)
	MM2VIS.bGCB_MDL			:=		IN_SY.tGCB_MDL.Di;		(* DI generator circuit breaker master demand lock (for closing other GCB to dead BB) *)
	MM2VIS.bGCB_MRC			:=		IN_SY.tGCB_MRC.Di;		(* DI generator circuit breaker master release close (to dead busbar) *)
	MM2VIS.bGCB_AGO			:=		IN_SY.tGCB_AGO.Di;		(* DI all other generator circuit breaker off *)
	MM2VIS.bGCB_RI			:=		IN_SY.tGCB_RI.Di;		(* DI generator circuit breaker reelase island *)
	MM2VIS.bGCB_OGP			:=		IN_SY.tGCB_OGP.Di OR IN_SY.bGCB_OGP_Bus;		(* DI generator circuit breaker other generator parallel *)
	MM2VIS.bGCB_DVM			:=		IN_SY.tGCB_DVM.Di;		(* DI voltage matching for synchronization *)
	MM2VIS.bGCB_DSY			:=		IN_SY.tGCB_DSY.Di;		(* DI generator circuit breaker demand synchronization (synchline) *)
//	MM2VIS.bF_N_DI_Inc		:=		IN_OP.tF_N_DI_Inc.Di;	(* DI synch.increase speed *)
//	MM2VIS.bF_N_DI_Dec		:=		IN_OP.tF_N_DI_Dec.Di;	(* DI synch.decrease speed *)
//	MM2VIS.bU_Gen_Inc		:=		IN_GC.tU_Gen_Inc.Di;	(* DI voltage adjustment external (increasing)*)
//	MM2VIS.bU_Gen_Dec		:=		IN_GC.tU_Gen_Dec.Di;	(* DI voltage adjustment external (decreasing)*)

	MM2VIS.bRdy_MSy			:=		OUT_SY.tRdy_MSy.Do;		(* DO engine ready    for MSY/GSY *)
	MM2VIS.bEng_Run_Sy		:=		OUT_SY.tEng_Run_Sy.Do;	(* DO engine rotating for MSY/GSY *)
	MM2VIS.bEng_Dem			:=		OUT_SY.tEng_Dem.Do;		(* DO engine demanded for MSY/GSY *)
	MM2VIS.bGCB_OpF			:=		OUT_SY.tGCB_OpF.Do;		(* DO alarm gcb opening failure *)
	MM2VIS.bGCB_EDC			:=		OUT_SY.tGCB_EDC.Do;		(* DO ESY demand lock all other cb's connected to dead busbar *)
	MM2VIS.bGCB_ESL			:=		OUT_SY.tGCB_ESL.Do;		(* DO ESY status gcb locked *)

//	MM2VIS.bImp_OpHour  	:= 		OUT_OP.tImp_OpHour.Do;	(* DO Impulse for operation hour counter *)
//	MM2VIS.bEng_Rdy_Rem 	:= 		OUT_OP.tEng_Rdy_Rem.Do;	(* DO Ready for Remote Operation *)
//	MM2VIS.bEng_Run 		:=		OUT_OP.tEng_Run.Do;		(* DO Engine in operation*)

	MM2VIS.bDemGenExcOff	:=		IN_SY.tDemGenExcOff.Di;	(* DI demand generator excitation off*)
	MM2VIS.bGenExcOff		:=		OUT_SY.tGenExcOff.Do;	(* DO generator excitation off*)

END_PROGRAM
```

### Program Logical/Synchronization/PermSY (IEC, version 4.10.0) - + PermanentMemory

- PermSYCyclic.st (not readable text: treated as protected, skipped)

- PermSYInit.st (not readable text: treated as protected, skipped)

#### PermSY.var
```iecst
VAR
	pm_Error : UINT;
	write_once : BOOL;
	pm_len : UDINT;
	ModulName : STRING[35];
	DatObjInfo_01 : DatObjInfo;
	pm_id : UDINT;
	pm_p : UDINT;
	bCreateDataObj : BOOL;
	perm_par_vers : UINT;
	DatObjRead_01 : DatObjRead;
	DatObjDelete_PermMem : DatObjDelete;
	DatObjCreate_01 : DatObjCreate;
	DatObjWrite_01 : DatObjWrite;
	ulChecksumOld : UDINT;
	ulPMPointer : UDINT;
	ulChkValue : UDINT;
	TON_WritePMEM : TON;
	ulChecksum : UDINT;
	bWriteDataObj : BOOL;
	TON_WarnDelay : TON;
	TON_BlockMinFileAge : TON; (*waiting time without file write after successful performed write*)
	bBlock_MinFileAge : BOOL := FALSE; (*pause the perm file write after each sucessful write*)
	iPM_WriteCnt : UDINT; (* *) (*old VarName: usPMWriteCnt*)
END_VAR
VAR CONSTANT
	ERR_NOERROR : UINT := 0;
END_VAR
VAR
	pmm : Perm_SY_Struct;
END_VAR
```

### Program Logical/Synchronization/ParSY (IEC, version 4.06.0) - + parameter handling

- perm_par.st (not readable text: treated as protected, skipped)

#### perm_par.var
```iecst
VAR
	tParaIntern : ParaHandler_typ; (*Connector type to perm_par*)
	tMM2ParaBase_ReadBack : MM2ParaBase_type; (*INTERNAL! V4.06 new readback structure for information from previous tasks*)
	bWriteDataObj : BOOL; (* TRUE=write data object module *)
	bDataObjLenErr : BOOL; (*Error occured in permem: data module size missmatch*)
	bCreateDataObj : BOOL; (* TRUE=create new data object *)
	bWriteOnce : BOOL; (* write permanent memory once *)
	DatObjCreate_01 : DatObjCreate; (* data object create *)
	DatObjInfoBak_02 : DatObjInfo; (* data object info *)
	DatObjDelete_01 : DatObjDelete; (* data object delete *)
	DatObjRead_01 : DatObjRead; (* data object read *)
	DatObjRead_02 : DatObjRead; (* manual initiated data object read *)
	DatObjWrite_01 : DatObjWrite; (* data object write *)
	DatObjDelete_02 : DatObjDelete; (* data object delete *)
	DatObjDelete_11 : DatObjDelete; (*Delete Backup File*)
	DatObjInfo_01 : DatObjInfo; (* data object info *)
	DatObjInfo_02 : DatObjInfo; (* data object info *)
	szModuleName : STRING[35]; (* module name of object *)
	szModuleNameBackup : STRING[35]; (* module name of posiibly created backup object *)
	DatObjCopy_01 : DatObjCopy;
	bCopyDataObj : BOOL;
	TON_WarnDelay : TON;
	TON_WritePMEM : TON; (* delay write permanent memory *)
	ulPMPointer : UDINT; (* adress of actual checksum value *)
	ulChecksum : UDINT; (* parameter checksum value *)
	pm_len : UDINT; (* permanent value lenght *)
	ulChecksumOld : UDINT; (* last vlaue of parameter checksum *)
	ulChkValue : UDINT; (* actual value of parameter pointer *)
	pm_id : UDINT; (* permanent value identifier *)
	pm_p : UDINT; (* permanent value pointer *)
	DatObjInfo_META : DatObjInfo;
	DatObjRead_META : DatObjRead;
	szMetaDataRaw : STRING[2000];
	szMetaData : ARRAY[0..4] OF STRING[35];
	szMetaDataVis : ARRAY[0..3] OF STRING[35];
	ssIndex : INT;
	ssCount : INT;
	ucMetaDataRaw : ARRAY[0..2000] OF USINT;
	ssCount2 : INT;
	szMetaDataFile : STRING[10];
	szText1 : STRING[20];
	pv_adr_IN_XX_tPB2MM : UDINT;
	pv_lng : UDINT;
	pv_lng_IN_XX_tPB2MM : UDINT;
	pv_lng_OUT_XX_tPB2MM : UDINT;
	szText2 : STRING[20];
	pv_adr_OUT_XX_tXX2PB : UDINT;
END_VAR
VAR CONSTANT
	ERR_NOERROR : UINT := 0;
END_VAR
VAR
	usPMWriteCnt : UINT;
	pm_Error : UDINT; (* permanent value error *) (* Deleted: pm : ParaMem_typ; permanent memory tags mathias, 22.8.11*)
	fun_Error : UDINT := 0; (*state > 0 = function error*)
	xLocalParaCheck : ParaCheckFUB; (*local function instance to check parameter values*)
	TON_ParaSetupOk : TON;
	bParaCheckSystemOk : BOOL;
	iDebug_ParaOkChecked : UDINT;
	bRestoreBackupDataObj : BOOL := FALSE;
	bRestoreDataObjContent : BOOL := FALSE;
	pm_id_backup : UDINT;
	pm_p_Backup : UDINT;
	DatObjCopy_02 : DatObjCopy;
	bDeleteBackupDataObj : BOOL := FALSE; (*Command to delete backup data module file on purpose*)
	bDebugPara : ARRAY[0..5] OF BOOL;
	ssIndex2 : INT;
	ssIndex3 : INT;
	ssIndex4 : INT;
	ssIndexVis : INT;
	szText : STRING[40];
	pv_adr_Para : UDINT;
	szParaSnippet : ARRAY[0..5] OF STRING[150];
	szParaIndex : STRING[10];
	slValue : DINT;
	iModuleDLD_ResetCount : INT;
	bDownloadDetected : BOOL;
	bFlagParaStructCopyWorking : BOOL; (*true, if cyclic para copying is active, 1 false cycle at every copy *)
	bStoreInitParaInDataObj : BOOL := FALSE;
	bTestflag : BOOL;
	bReadOutMETA_Once : BOOL;
	tParaCheck_iPvAdress : ARRAY[0..5] OF UDINT;
	tParaCheck_iPvLengt : ARRAY[0..5] OF UDINT;
	tParaCheck_rPvValue : ARRAY[0..5] OF REAL;
	tParaCheck_rRangeMIN : ARRAY[0..5] OF REAL;
	tParaCheck_rRangeMAX : ARRAY[0..5] OF REAL;
	tParaCheck_szPvName : ARRAY[0..5] OF STRING[35];
	ssFormatDetected : INT;
	szMetaDataPart : STRING[150];
	szFullTaskName : STRING[35];
	szFullMetaModuleName : STRING[35];
	debugLen : INT;
	debugSize : INT := 0;
	strcat_adr1 : UDINT;
	strcat_adr2 : UDINT;
	ssIndexTN : INT;
	bAlternate : BOOL;
	n : INT;
	iAlternateChecksum : DINT;
	iAlternateChecksumOld : DINT;
	ulDebugChkValue : ARRAY[0..999] OF UDINT;
	Adr1 : UDINT;
	Adr2 : UDINT;
	usPMWriteCntStepsize : UINT := 1; (*different step sizes to help debug*)
	usPMWriteCntXOR : UINT;
	usPMWriteCntAltSum : UINT;
	ulAdrPM : UDINT;
	usChkValuePM : USINT;
	ulAdrPara : UDINT;
	ulPara_len : UDINT;
	usChkValuePara : USINT;
	iDebugCountPMDifferences : DINT := 0;
	bEngineRunDetected : BOOL; (*detection status bit autocommand 100 /101  for engine run state*)
	ucMetaDataDebugInfoLine : ARRAY[0..24] OF STRING[80];
	ssIndexMand : INT := 0;
	szMetaDataMand : STRING[35];
	iMyErrorInfo_Autoreset : DINT; (*internal autoreset counter*)
	ssIndex_Version : INT; (*internal*)
	ssIndex_BU : INT; (*internal*)
	ssIndex_BU2 : INT; (*internal*)
END_VAR
```

### Program Logical/Synchronization/LV_GCB (IEC) - LV GCB communication

#### LV_GCB_Cyclic.st - Cyclic
```iecst
(*******************************************************************************
AGGR: Modbus RTU connection to LV GCB  (cyclic)

This code is confidential and proprietary to the INNIO Company.
It may not be used in any form, or reproduced in any manner, without the express
written permission of the INNIO Company.
Copyright, INNIO Company, 2023

Customized modifications: -
------------------------

History:
-------
V4.13	14-11-2023	Hohensinner	created

Instructions for use:
--------------------
Caution!
- X20CS1030_xxx_xx_GCB should not be in "cyclic stream" mode, instead it should be set to "stream".
- Also the modules name must be ending with "_GCB" to be found in the init part.

Outstandings:
------------
*******************************************************************************)

PROGRAM _CYCLIC

	(** 1: waiting for parasetup okay *)
	xTON_ParaSetup_Ok(IN:= TRUE AND NOT bError_Conf, PT:= tiParaSetup_Ok);
	IF NOT xTON_ParaSetup_Ok.Q OR bDeactivate_Task OR DiagCpuIsSimulated() THEN RETURN; END_IF

	(** 2: running the modbus master *)
	xTON_Rel_MBMaster(IN:= xTON_ParaSetup_Ok.Q, PT:=tiRel_MBMaster);
	xMBDO_Master[0].bEnable	:=	xTON_Rel_MBMaster.Q;
	xMBDO_Master[0]();

	(** 3: State Machine of LV GCB connection *)
	CASE eState_GCB OF
		_GCB_INIT:
			eState_GCB := _GCB_TRY_ABB;
		_GCB_TRY_ABB:
			(* Init *)
			IF bInit THEN
				tSlave[0].tLine[0].tIF.bExec	:=	TRUE;	//make first contact
			END_IF
			(* Wait *)
			xWAIT(IN:=1);
			(* Exit *)
			IF xWAIT.Q THEN
				IF 	NOT tSlave[0].tLine[0].tIF.bExec AND tSlave[0].tLine[0].tIF.iStatus = 0 THEN
					eState_GCB := _GCB_IDLE;
					MM2VIS.tGCB[1].iType	:= 1;
				ELSIF tSlave[0].tLine[0].tIF.bExec AND tSlave[0].tLine[0].tIF.iStatus <> ERR_FUB_BUSY THEN
					eState_GCB := _GCB_TRY_SE;
					tSlave[0].tLine[0].tIF.bExec	:=	FALSE;	//end first contact
				END_IF
			END_IF
		_GCB_TRY_SE:
			(* Init *)
			IF bInit THEN
				tSlave[1].tLine[0].tIF.bExec	:=	TRUE;	//make first contact
			END_IF
			(* Wait *)
			xWAIT(IN:=1);
			(* Exit *)
			IF xWAIT.Q THEN
				IF 	NOT tSlave[1].tLine[0].tIF.bExec AND tSlave[1].tLine[0].tIF.iStatus = 0 THEN
					eState_GCB := _GCB_IDLE;
					MM2VIS.tGCB[1].iType	:= 2;
				ELSIF tSlave[1].tLine[0].tIF.bExec AND tSlave[1].tLine[0].tIF.iStatus <> ERR_FUB_BUSY THEN
					eState_GCB := _GCB_WAIT;
					tSlave[1].tLine[0].tIF.bExec	:=	FALSE;	//end first contact
				END_IF
			END_IF
		_GCB_WAIT:
			(* Wait *)
			xWAIT(IN:=100);
			(* Exit *)
			IF xWAIT.Q THEN
				eState_GCB := _GCB_TRY_ABB;
			END_IF
		_GCB_CALC:
			FOR i:=0 TO 60 DO
				rFactors := 0.4 + UINT_TO_REAL(i) * 0.01;
				IF VIS2MM.tGCB[1].rI_GenNom * 1.1 <= rFactors * MM2VIS.tGCB[1].rI_Nom THEN
					EXIT;
				END_IF
			END_FOR
			VIS2MM.tGCB[1].rI1	:=	MM2VIS.tGCB[1].rI_Nom * rFactors;
			IF bSE THEN
				VIS2MM.tGCB[1].rt1	:=	1;
			ELSIF bABB THEN
				VIS2MM.tGCB[1].rt1	:=	3;
			END_IF
			VIS2MM.tGCB[1].rI2	:=	MM2VIS.tGCB[1].rI_Nom * 2;
			VIS2MM.tGCB[1].rt2	:=	0.3;
			VIS2MM.tGCB[1].rI3	:=	MM2VIS.tGCB[1].rI_Nom * 10;
			eState_GCB := _GCB_IDLE;
		_ABB_LOAD:
			(* Init *)
			IF bInit THEN
				VIS2MM.tGCB[1].rI_GenNom := Para.rI_GenNom[1];
				tSlave[0].tLine[6].tIF.bExec	:=	TRUE;
				tSlave[0].tLine[7].tIF.bExec	:=	TRUE;
				tSlave[0].tLine[8].tIF.bExec	:=	TRUE;
				tSlave[0].tLine[12].tIF.bExec	:=	TRUE;
			END_IF
			(* Wait *)
			xWAIT(IN:=1);
			MM2VIS.tGCB[1].rLoad	:=	BOOL_TO_REAL(NOT tSlave[0].tLine[6].tIF.bExec)/4
									+	BOOL_TO_REAL(NOT tSlave[0].tLine[7].tIF.bExec)/4
									+	BOOL_TO_REAL(NOT tSlave[0].tLine[8].tIF.bExec)/4
									+	BOOL_TO_REAL(NOT tSlave[0].tLine[12].tIF.bExec)/4;
			(* Exit *)
			IF NOT tSlave[0].tLine[6].tIF.bExec AND NOT tSlave[0].tLine[7].tIF.bExec AND
				NOT tSlave[0].tLine[8].tIF.bExec AND NOT tSlave[0].tLine[12].tIF.bExec AND xWAIT.Q THEN
				MM2VIS.tGCB[1].rI_Nom			:=	UINT_TO_REAL(tSlave[0].tLine[12].tIF.iData[0]);
				VIS2MM.tGCB[1].rI1				:=	MM2VIS.tGCB[1].rI_Nom * UINT_TO_REAL(tSlave[0].tLine[6].tIF.iData[1])/1000;
				VIS2MM.tGCB[1].rt1				:=	UINT_TO_REAL(tSlave[0].tLine[6].tIF.iData[2])/100;
				VIS2MM.tGCB[1].rI2				:=	MM2VIS.tGCB[1].rI_Nom * UINT_TO_REAL(tSlave[0].tLine[7].tIF.iData[1])/100;
				VIS2MM.tGCB[1].rt2				:=	UINT_TO_REAL(tSlave[0].tLine[7].tIF.iData[2])/100;
				VIS2MM.tGCB[1].rI3				:=	MM2VIS.tGCB[1].rI_Nom * UINT_TO_REAL(tSlave[0].tLine[8].tIF.iData[1])/100;
				eState_GCB := _ABB_READ;
			END_IF
		_ABB_READ:
			(* Init *)
			IF bInit THEN
				tSlave[0].tLine[0].tIF.bExec	:=	TRUE;
				tSlave[0].tLine[2].tIF.bExec	:=	TRUE;
				tSlave[0].tLine[3].tIF.bExec	:=	TRUE;
				tSlave[0].tLine[4].tIF.bExec	:=	TRUE;
				tSlave[0].tLine[11].tIF.bExec	:=	TRUE;
				tSlave[0].tLine[12].tIF.bExec	:=	TRUE;
			END_IF
			(* Wait *)
			xWAIT(IN:=1);
			(* Exit *)
			IF 	NOT tSlave[0].tLine[0].tIF.bExec AND
				NOT tSlave[0].tLine[2].tIF.bExec AND
				NOT tSlave[0].tLine[3].tIF.bExec AND
				NOT tSlave[0].tLine[4].tIF.bExec AND
				NOT tSlave[0].tLine[11].tIF.bExec AND
				NOT tSlave[0].tLine[12].tIF.bExec AND xWAIT.Q THEN
				MM2VIS.tGCB[1].rWear			:=	UINT_TO_REAL(tSlave[0].tLine[0].tIF.iData[0])/65000;
				MM2VIS.tGCB[1].iNumOp			:=	UINT_TO_DINT(tSlave[0].tLine[0].tIF.iData[1]);
				MM2VIS.tGCB[1].iNumPT			:=	UINT_TO_DINT(tSlave[0].tLine[0].tIF.iData[3]);
				MM2VIS.tGCB[1].rI_Act_L1		:=	(UINT_TO_REAL(tSlave[0].tLine[2].tIF.iData[0])+UINT_TO_REAL(tSlave[0].tLine[2].tIF.iData[1])*65536)/10;
				MM2VIS.tGCB[1].rI_Act_L2		:=	(UINT_TO_REAL(tSlave[0].tLine[2].tIF.iData[2])+UINT_TO_REAL(tSlave[0].tLine[2].tIF.iData[3])*65536)/10;
				MM2VIS.tGCB[1].rI_Act_L3		:=	(UINT_TO_REAL(tSlave[0].tLine[2].tIF.iData[4])+UINT_TO_REAL(tSlave[0].tLine[2].tIF.iData[5])*65536)/10;
				MM2VIS.tGCB[1].rU_Act			:=	UINT_TO_REAL(tSlave[0].tLine[3].tIF.iData[0])/10/3
												+	UINT_TO_REAL(tSlave[0].tLine[3].tIF.iData[1])/10/3
												+	UINT_TO_REAL(tSlave[0].tLine[3].tIF.iData[2])/10/3;
				MM2VIS.tGCB[1].rU_Nom			:=	UINT_TO_REAL(tSlave[0].tLine[4].tIF.iData[0]);
				MM2VIS.tGCB[1].bClosed			:=	tSlave[0].tLine[11].tIF.iData[0].0;
				MM2VIS.tGCB[1].bRacked			:=	tSlave[0].tLine[11].tIF.iData[0].1;
				MM2VIS.tGCB[1].bFail			:=	tSlave[0].tLine[11].tIF.iData[0].13
												OR	tSlave[0].tLine[11].tIF.iData[0].7
												OR NOT tSlave[0].tLine[11].tIF.iData[0].8
												OR	tSlave[0].tLine[11].tIF.iData[0].10
												OR	tSlave[0].tLine[11].tIF.iData[0].5;
				MM2VIS.tGCB[1].rI_Nom			:=	UINT_TO_REAL(tSlave[0].tLine[12].tIF.iData[0]);
				bABB_Remote						:= tSlave[0].tLine[11].tIF.iData[0].8;
				eState_GCB := _GCB_IDLE;
			END_IF
		_ABB_SAVE_OPEN:
			(* Init *)
			IF bInit THEN
				tSlave[0].tLine[13].tIF				:=	tIF_ABB_Open;
				MM2VIS.tGCB[1].rSave				:=	0.33;
			END_IF
			(* Wait *)
			xWAIT(IN:=1);
			(* Exit *)
			IF NOT tSlave[0].tLine[13].tIF.bExec AND xWAIT.Q THEN
				eState_GCB := _ABB_SAVE_DATA;
			END_IF
		_ABB_SAVE_DATA:
			(* Init *)
			IF bInit THEN																												//LOW	HIGH	STEP
				tSlave[0].tLine[14].tIF.iData[0]	:=	LIMIT(REAL_TO_UINT(VIS2MM.tGCB[1].rI1/MM2VIS.tGCB[1].rI_Nom*1000),400,1000);	//400	1000	1
				tSlave[0].tLine[14].tIF.iData[1]	:=	LIMIT(REAL_TO_UINT(VIS2MM.tGCB[1].rt1),3,144)*100;								//300	14400	100
				tSlave[0].tLine[9].tIF.iData[0]		:=	LIMIT(REAL_TO_UINT(VIS2MM.tGCB[1].rI2/MM2VIS.tGCB[1].rI_Nom*10),6,100)*10;		//60	1000	10
				tSlave[0].tLine[9].tIF.iData[1]		:=	LIMIT(REAL_TO_UINT(VIS2MM.tGCB[1].rt2*100),5,80);								//5		80		1
				tSlave[0].tLine[10].tIF.iData[0]	:=	LIMIT(REAL_TO_UINT(VIS2MM.tGCB[1].rI3/MM2VIS.tGCB[1].rI_Nom*10),15,150)*10;		//150	1500	10
				tSlave[0].tLine[14].tIF.bExec		:=	TRUE;
				tSlave[0].tLine[9].tIF.bExec		:=	TRUE;
				tSlave[0].tLine[10].tIF.bExec		:=	TRUE;
				MM2VIS.tGCB[1].rSave				:=	0.66;
			END_IF
			(* Wait *)
			xWAIT(IN:=1);
			(* Exit *)
			IF NOT tSlave[0].tLine[14].tIF.bExec AND NOT tSlave[0].tLine[9].tIF.bExec AND NOT tSlave[0].tLine[10].tIF.bExec AND xWAIT.Q THEN
				eState_GCB := _ABB_SAVE_CLOSE;
			END_IF
		_ABB_SAVE_CLOSE:
			(* Init *)
			IF bInit THEN
				tSlave[0].tLine[13].tIF		:=	tIF_ABB_Close;
			END_IF
			(* Wait *)
			xWAIT(IN:=1);
			(* Exit *)
			IF NOT tSlave[0].tLine[13].tIF.bExec AND xWAIT.Q THEN
				eState_GCB := _ABB_LOAD;
				MM2VIS.tGCB[1].rSave				:=	1.00;
			END_IF
		_SE_LOAD:
			(* Init Load *)
			IF bInit THEN
				VIS2MM.tGCB[1].rI_GenNom := Para.rI_GenNom[1];
				tSlave[1].tLine[4].tIF.bExec	:=	TRUE;	//to load I_Nom
				tSlave[1].tLine[6].tIF.bExec	:=	TRUE;
				tSlave[1].tLine[7].tIF.bExec	:=	TRUE;
				tSlave[1].tLine[8].tIF.bExec	:=	TRUE;
			END_IF
			(* Wait Load *)
			xWAIT(IN:=1);
			MM2VIS.tGCB[1].rLoad	:=	BOOL_TO_REAL(NOT tSlave[1].tLine[4].tIF.bExec)/4
									+	BOOL_TO_REAL(NOT tSlave[1].tLine[6].tIF.bExec)/4
									+	BOOL_TO_REAL(NOT tSlave[1].tLine[7].tIF.bExec)/4
									+	BOOL_TO_REAL(NOT tSlave[1].tLine[8].tIF.bExec)/4;
			(* Exit Load *)
			IF NOT tSlave[1].tLine[4].tIF.bExec AND NOT tSlave[1].tLine[6].tIF.bExec AND NOT tSlave[1].tLine[7].tIF.bExec AND NOT tSlave[1].tLine[8].tIF.bExec AND xWAIT.Q THEN
				MM2VIS.tGCB[1].rI_Nom	:=	UINT_TWO_REAL(tSlave[1].tLine[4].tIF.iData[2],tSlave[1].tLine[4].tIF.iData[3]);
				VIS2MM.tGCB[1].rI1	:=	UINT_TWO_REAL(tSlave[1].tLine[6].tIF.iData[0],tSlave[1].tLine[6].tIF.iData[1]);
				VIS2MM.tGCB[1].rt1	:=	UINT_TWO_REAL(tSlave[1].tLine[6].tIF.iData[2],tSlave[1].tLine[6].tIF.iData[3]);
				rFactor_Isd			:=	UINT_TWO_REAL(tSlave[1].tLine[7].tIF.iData[0],tSlave[1].tLine[7].tIF.iData[1]);
				VIS2MM.tGCB[1].rI2	:=	rFactor_Isd*VIS2MM.tGCB[1].rI1;
				VIS2MM.tGCB[1].rt2	:=	UINT_TWO_REAL(tSlave[1].tLine[7].tIF.iData[2],tSlave[1].tLine[7].tIF.iData[3]);
				rFactor_Ii			:=	UINT_TWO_REAL(tSlave[1].tLine[8].tIF.iData[1],tSlave[1].tLine[8].tIF.iData[2]);
				VIS2MM.tGCB[1].rI3	:=	rFactor_Ii*MM2VIS.tGCB[1].rI_Nom;
				eState_GCB := _SE_READ;
			END_IF
		_SE_READ:
			(* Init Read *)
			IF bInit THEN
				tSlave[1].tLine[0].tIF.bExec	:=	TRUE;
				tSlave[1].tLine[1].tIF.bExec	:=	TRUE;
				tSlave[1].tLine[2].tIF.bExec	:=	TRUE;
				tSlave[1].tLine[3].tIF.bExec	:=	TRUE;
				tSlave[1].tLine[4].tIF.bExec	:=	TRUE;
				tSlave[1].tLine[5].tIF.bExec	:=	TRUE;
//				tSlave[1].tLine[9].tIF.bExec	:=	TRUE;		//falls SE racked in / out IO interface besitzt aktivieren
			END_IF
			(* Wait Read *)
			xWAIT(IN:=1);
			(* Exit Read *)
			IF 	NOT tSlave[1].tLine[0].tIF.bExec AND
				NOT tSlave[1].tLine[1].tIF.bExec AND
				NOT tSlave[1].tLine[2].tIF.bExec AND
				NOT tSlave[1].tLine[3].tIF.bExec AND
				NOT tSlave[1].tLine[4].tIF.bExec AND
				NOT tSlave[1].tLine[5].tIF.bExec AND
				NOT tSlave[1].tLine[9].tIF.bExec AND xWAIT.Q THEN
				MM2VIS.tGCB[1].iNumOp			:=	UDINT_TO_DINT(UINT_TWO_UDINT(tSlave[1].tLine[0].tIF.iData[0],tSlave[1].tLine[0].tIF.iData[1]));
				MM2VIS.tGCB[1].iNumPT			:=	UDINT_TO_DINT(UINT_TWO_UDINT(tSlave[1].tLine[0].tIF.iData[2],tSlave[1].tLine[0].tIF.iData[3]));
				MM2VIS.tGCB[1].rI_Act_L1		:=	UINT_TWO_REAL(tSlave[1].tLine[2].tIF.iData[0],tSlave[1].tLine[2].tIF.iData[1]);
				MM2VIS.tGCB[1].rI_Act_L2		:=	UINT_TWO_REAL(tSlave[1].tLine[2].tIF.iData[2],tSlave[1].tLine[2].tIF.iData[3]);
				MM2VIS.tGCB[1].rI_Act_L3		:=	UINT_TWO_REAL(tSlave[1].tLine[2].tIF.iData[4],tSlave[1].tLine[2].tIF.iData[5]);
				MM2VIS.tGCB[1].rU_Act			:=	UINT_TWO_REAL(tSlave[1].tLine[3].tIF.iData[0],tSlave[1].tLine[3].tIF.iData[1]);
				MM2VIS.tGCB[1].rU_Nom			:=	UINT_TWO_REAL(tSlave[1].tLine[4].tIF.iData[0],tSlave[1].tLine[4].tIF.iData[1]);
				MM2VIS.tGCB[1].rI_Nom			:=	UINT_TWO_REAL(tSlave[1].tLine[4].tIF.iData[2],tSlave[1].tLine[4].tIF.iData[3]);
				MM2VIS.tGCB[1].rWear			:=	UINT_TWO_REAL(tSlave[1].tLine[5].tIF.iData[0],tSlave[1].tLine[5].tIF.iData[1]);
				MM2VIS.tGCB[1].bClosed			:=	tSlave[1].tLine[1].tIF.iData[1].0;
				MM2VIS.tGCB[1].bRacked			:=	tSlave[1].tLine[9].tIF.iData[0].9;
				eState_GCB := _GCB_IDLE;
			END_IF
		_SE_SAVE_CHECK:												 //Check if no session is open
			(* Init Check *)
			IF bInit THEN
				tSlave[1].tLine[11].tIF.bExec		:=	TRUE;
				MM2VIS.tGCB[1].rSave				:=	0.1;
			END_IF
			(* Wait Check *)
			xWAIT(IN:=1);
			(* Exit Check *)
			IF NOT tSlave[1].tLine[11].tIF.bExec AND xWAIT.Q THEN
				IF (tSlave[1].tLine[11].tIF.iData[3] <> 0 OR tSlave[1].tLine[11].tIF.iData[4] <> 0) AND tSlave[1].tLine[11].tIF.iData[0]<>1933 THEN
					iSessionKey0 := tSlave[1].tLine[11].tIF.iData[3];
					iSessionKey1 := tSlave[1].tLine[11].tIF.iData[4];
					eState_GCB := _SE_SAVE_CLOSE_OLD;
				ELSE
					eState_GCB := _SE_SAVE_OPEN;
				END_IF
			END_IF
		_SE_SAVE_CLOSE_OLD:								//close old session
			(* Init Close *)
			IF bInit THEN
				tSlave[1].tLine[10].tIF 			:=	tIF_Session_Close;
				tSlave[1].tLine[10].tIF.iData[6]	:=	iSessionKey0;
				tSlave[1].tLine[10].tIF.iData[7]	:=	iSessionKey1;
				MM2VIS.tGCB[1].rSave				:=	0.2;
			END_IF
			(* Wait Close *)
			xWAIT(IN:=1);
			(* Exit Close *)
			IF NOT tSlave[1].tLine[10].tIF.bExec AND xWAIT.Q THEN
				eState_GCB := _SE_SAVE_OPEN;
			END_IF
		_SE_SAVE_OPEN:										//open new session
			(* Init Open *)
			IF bInit THEN
				tSlave[1].tLine[10].tIF 			:=	tIF_Session_Open;
				MM2VIS.tGCB[1].rSave				:=	0.3;
			END_IF
			(* Wait Open *)
			xWAIT(IN:=1);
			(* Exit Open *)
			IF NOT tSlave[1].tLine[10].tIF.bExec AND xWAIT.Q THEN
				eState_GCB := _SE_SAVE_ID;
			END_IF
		_SE_SAVE_ID:										//ask for new session ID
			(* Init ID *)
			IF bInit THEN
				tSlave[1].tLine[11].tIF.bExec		:=	TRUE;
				MM2VIS.tGCB[1].rSave				:=	0.4;
			END_IF
			(* Wait ID *)
			xWAIT(IN:=1);
			(* Exit ID *)
			IF NOT tSlave[1].tLine[11].tIF.bExec THEN
				IF tSlave[1].tLine[11].tIF.iData[1] = 0 AND tSlave[1].tLine[11].tIF.iData[2] = 4 AND xWAIT.Q THEN
					iSessionKey0 := tSlave[1].tLine[11].tIF.iData[3];
					iSessionKey1 := tSlave[1].tLine[11].tIF.iData[4];
					eState_GCB := _SE_SAVE_DATA1;
				ELSE
					iSessionKey0 := tSlave[1].tLine[11].tIF.iData[3];
					iSessionKey1 := tSlave[1].tLine[11].tIF.iData[4];
					eState_GCB := _SE_SAVE_CLOSE_OLD;
				END_IF
			END_IF
		_SE_SAVE_DATA1:											//change Dataset 1
			(* Init Data1 *)
			IF bInit THEN
				tSlave[1].tLine[10].tIF				:=	tIF_Session_Change1;
				tSlave[1].tLine[10].tIF.iData[6]	:=	iSessionKey0;
				tSlave[1].tLine[10].tIF.iData[7]	:=	iSessionKey1;
				rTemp := STEP(VIS2MM.tGCB[1].rI1,0.1);
				brsmemcpy(ADR(tSlave[1].tLine[10].tIF.iData[10]),ADR(rTemp)+2,2);
				brsmemcpy(ADR(tSlave[1].tLine[10].tIF.iData[11]),ADR(rTemp),2);
				rTemp := LIMIT(STEP(VIS2MM.tGCB[1].rt1,0.5),0.5,24.0);
				brsmemcpy(ADR(tSlave[1].tLine[10].tIF.iData[12]),ADR(rTemp)+2,2);
				brsmemcpy(ADR(tSlave[1].tLine[10].tIF.iData[13]),ADR(rTemp),2);
				MM2VIS.tGCB[1].rSave				:=	0.5;
			END_IF
			(* Wait Data1 *)
			xWAIT(IN:=1);
			(* Exit Data1 *)
			IF NOT tSlave[1].tLine[10].tIF.bExec AND xWAIT.Q THEN
				eState_GCB := _SE_SAVE_DATA2;
			END_IF
		_SE_SAVE_DATA2:											//change Dataset 2
			(* Init Data2 *)
			IF bInit THEN
				tSlave[1].tLine[10].tIF				:=	tIF_Session_Change2;
				tSlave[1].tLine[10].tIF.iData[6]	:=	iSessionKey0;
				tSlave[1].tLine[10].tIF.iData[7]	:=	iSessionKey1;
				rTemp := LIMIT(STEP(VIS2MM.tGCB[1].rI2/VIS2MM.tGCB[1].rI1,0.1),1.5,10.0);
				brsmemcpy(ADR(tSlave[1].tLine[10].tIF.iData[10]),ADR(rTemp)+2,2);
				brsmemcpy(ADR(tSlave[1].tLine[10].tIF.iData[11]),ADR(rTemp),2);
				rTemp := LIMIT(STEP(VIS2MM.tGCB[1].rt2,0.1),0.0,0.4);
				brsmemcpy(ADR(tSlave[1].tLine[10].tIF.iData[12]),ADR(rTemp)+2,2);
				brsmemcpy(ADR(tSlave[1].tLine[10].tIF.iData[13]),ADR(rTemp),2);
				MM2VIS.tGCB[1].rSave				:=	0.6;
			END_IF
			(* Wait Data2 *)
			xWAIT(IN:=1);
			(* Exit Data2 *)
			IF NOT tSlave[1].tLine[10].tIF.bExec AND xWAIT.Q THEN
				eState_GCB := _SE_SAVE_DATA3;
			END_IF
		_SE_SAVE_DATA3:										//change Dataset 3
			(* Init Data3 *)
			IF bInit THEN
				tSlave[1].tLine[10].tIF				:=	tIF_Session_Change3;
				tSlave[1].tLine[10].tIF.iData[6]	:=	iSessionKey0;
				tSlave[1].tLine[10].tIF.iData[7]	:=	iSessionKey1;
				rTemp := LIMIT(STEP(VIS2MM.tGCB[1].rI3/MM2VIS.tGCB[1].rI_Nom,0.1),2.0,15.0);
				brsmemcpy(ADR(tSlave[1].tLine[10].tIF.iData[9]),ADR(rTemp)+2,2);
				brsmemcpy(ADR(tSlave[1].tLine[10].tIF.iData[10]),ADR(rTemp),2);
				MM2VIS.tGCB[1].rSave				:=	0.7;
			END_IF
			(* Wait Data3 *)
			xWAIT(IN:=1);
			(* Exit Data3 *)
			IF NOT tSlave[1].tLine[10].tIF.bExec AND xWAIT.Q THEN
				eState_GCB := _SE_SAVE_APPLY;
			END_IF
		_SE_SAVE_APPLY:										//apply changes
			(* Init Apply *)
			IF bInit THEN
				tSlave[1].tLine[10].tIF				:=	tIF_Session_Apply;
				tSlave[1].tLine[10].tIF.iData[6]	:=	iSessionKey0;
				tSlave[1].tLine[10].tIF.iData[7]	:=	iSessionKey1;
				MM2VIS.tGCB[1].rSave				:=	0.8;
			END_IF
			(* Wait Apply *)
			xWAIT(IN:=1);
			(* Exit Apply *)
			IF NOT tSlave[1].tLine[10].tIF.bExec AND xWAIT.Q THEN
				eState_GCB := _SE_SAVE_CLOSE;
			END_IF
		_SE_SAVE_CLOSE:										//close session
			(* Init Close *)
			IF bInit THEN
				tSlave[1].tLine[10].tIF 			:=	tIF_Session_Close;
				tSlave[1].tLine[10].tIF.iData[6]	:=	iSessionKey0;
				tSlave[1].tLine[10].tIF.iData[7]	:=	iSessionKey1;
				MM2VIS.tGCB[1].rSave				:=	0.9;
			END_IF
			(* Wait Close *)
			xWAIT(IN:=1);
			(* Exit Close *)
			IF NOT tSlave[1].tLine[10].tIF.bExec AND xWAIT.Q THEN
				eState_GCB := _SE_SAVE_CLOSE_CHECK;
			END_IF
		_SE_SAVE_CLOSE_CHECK:								 //Check if session is closed
			(* Init Check *)
			IF bInit THEN
				tSlave[1].tLine[11].tIF.bExec		:=	TRUE;
			END_IF
			(* Wait Check *)
			xWAIT(IN:=25);
			(* Exit Check *)
			IF NOT tSlave[1].tLine[11].tIF.bExec AND xWAIT.Q THEN
				IF tSlave[1].tLine[11].tIF.iData[0] = 1933 THEN
					eState_GCB := _SE_LOAD;
					MM2VIS.tGCB[1].rSave				:=	1.0;
				END_IF
			END_IF
		_GCB_CLEAR:
			MM2VIS.tGCB[1].iNumOp		:=	0;
			MM2VIS.tGCB[1].iNumPT		:=	0;
			MM2VIS.tGCB[1].rI_Act_L1	:=	0;
			MM2VIS.tGCB[1].rI_Act_L2	:=	0;
			MM2VIS.tGCB[1].rI_Act_L3	:=	0;
			MM2VIS.tGCB[1].rU_Act		:=	0;
			MM2VIS.tGCB[1].rU_Nom		:=	0;
			MM2VIS.tGCB[1].rI_Nom		:=	0;
			MM2VIS.tGCB[1].rWear		:=	0;
			MM2VIS.tGCB[1].bClosed		:=	0;
			MM2VIS.tGCB[1].bRacked		:=	0;
			MM2VIS.tGCB[1].bFail		:=	0;
			VIS2MM.tGCB[1].rI1			:=	0;
			VIS2MM.tGCB[1].rt1			:=	0;
			VIS2MM.tGCB[1].rI2			:=	0;
			VIS2MM.tGCB[1].rt2			:=	0;
			VIS2MM.tGCB[1].rI3			:=	0;

			IF bSE THEN		eState_GCB	:=	_SE_LOAD;
			ELSIF bABB THEN	eState_GCB	:=	_ABB_LOAD;
			ELSE			eState_GCB	:=	_GCB_IDLE;
			END_IF
		_GCB_IDLE:
			(* Wait Idle *)
			xWAIT(IN:=100);
			bABB	:=	MM2VIS.tGCB[1].iType = 1;
			bSE		:=	MM2VIS.tGCB[1].iType = 2;
			IF xWAIT.CNT > 30 THEN
				MM2VIS.tGCB[1].rSave	:= 0.0;
				MM2VIS.tGCB[1].rLoad	:= 0.0;
			END_IF
			(* Exit Idle *)
			IF bClear THEN
				bClear		:=	FALSE;
				eState_GCB	:=	_GCB_CLEAR;
			ELSIF VIS2MM.tGCB[1].bCalc THEN
				VIS2MM.tGCB[1].bCalc := FALSE;
				eState_GCB := _GCB_CALC;
			ELSIF VIS2MM.tGCB[1].bSave THEN
				VIS2MM.tGCB[1].bSave := FALSE;
				IF xOpMode.Stop THEN
					IF bSE THEN		eState_GCB := _SE_SAVE_CHECK; END_IF
					IF bABB AND bABB_Remote THEN	eState_GCB := _ABB_SAVE_OPEN; END_IF
				END_IF
			ELSIF VIS2MM.tGCB[1].bLoad THEN
				VIS2MM.tGCB[1].bLoad := FALSE;
				IF bSE THEN		eState_GCB := _SE_LOAD; END_IF
				IF bABB THEN	eState_GCB := _ABB_LOAD; END_IF
			ELSIF xWAIT.Q THEN
				IF bSE THEN		eState_GCB := _SE_READ; END_IF
				IF bABB THEN	eState_GCB := _ABB_READ; END_IF

			END_IF
	END_CASE

	(** 4: State Machine Helper *)
	IF eState_GCB <> eState_GCB_Old THEN
		bInit := TRUE;						//trigger init routine if state changed
		xWAIT(IN:=0);						//reset cyclic timer for new state
		xTIMEOUT(IN:=0);					//reset time out counter for new state;
		eState_GCB_Old := eState_GCB;
	ELSE
		bInit := FALSE;						//disable init routine after first run trough
		xTIMEOUT(IN:=1000);
		IF xTIMEOUT.Q THEN
			eState_GCB_TO	:=	eState_GCB;
			eState_GCB		:=	_GCB_IDLE;
		END_IF
	END_IF
	IF MM2VIS.tGCB[1].iType <> iType_Old THEN
		iType_Old	:=	MM2VIS.tGCB[1].iType;
		bClear	:=	TRUE;
	END_IF

	(** 5: Error Diagnostics *)
	IF bABB THEN
		MM2VIS.tGCB[1].iError	:=	xMBDO_Master[0].iLog[0];
	ELSIF bSE THEN
		MM2VIS.tGCB[1].iError	:=	xMBDO_Master[0].iLog[1];
	END_IF
	memcpy(ADR(MM2VIS.tGCB[1].iState),ADR(eState_GCB),2);

	(** 6: Operating Messages and Warnings *)
	(** 6.1: B9085 Parameters saved to the GCB *)
	xTOF_ParaSaved_5s.IN	:=	(bSE AND tSlave[1].tLine[11].tIF.iData[0] = 1933 AND eState_GCB_Old = _SE_SAVE_CLOSE_CHECK)
							OR	(bABB AND tSlave[0].tLine[13].tIF.iStatus = 0 AND eState_GCB_Old = _ABB_SAVE_CLOSE);
	xTOF_ParaSaved_5s.PT	:=	T#5s;
	xTOF_ParaSaved_5s();
	bB9085_GCB_ParaSaved := xTOF_ParaSaved_5s.Q;
	(** 6.2: W9382 GCB contact wear over 80% *)
	IF EDGEPOS(MM2VIS.tGCB[1].rWear >= 0.80) THEN
		bW9382_GCB_Wear80	:=	TRUE;
	END_IF
	IF IN_SY.tAB2SY.bResetWarning THEN
		bW9382_GCB_Wear80	:=	FALSE;
	END_IF
	(** 6.3: W9383 GCB contact wear over 95% *)
	bW9383_GCB_Wear95	:=	MM2VIS.tGCB[1].rWear >= 0.95;

END_PROGRAM
```

#### LV_GCB_Init.st - Init
```iecst
(*******************************************************************************
AGGR: Modbus RTU connection to LV GCB  (init)

This code is confidential and proprietary to the INNIO Company.
It may not be used in any form, or reproduced in any manner, without the express
written permission of the INNIO Company.
Copyright, INNIO Company, 2023

Customized modifications: -
------------------------

History:
-------
V4.13	21-11-2023	Hohensinner	created

Instructions for use:
--------------------
Caution!
- X20CS1030_xxx_xx_GCB should not be in "cyclic stream" mode, instead it should be set to "stream".
- Also the modules name must be ending with "_GCB" to be found in the init part.

Outstandings:
------------
*******************************************************************************)

PROGRAM _INIT
	(** 1: Don't execute task if ARsim is active *)
	IF DiagCpuIsSimulated() THEN
		RETURN;
	END_IF

	(** 2: get name and path of configured X20CS1030_xxx_xx_GCB module *)
	(** 2.1: get information about configured modules *)
	xDiagCreateInfo.enable		:= TRUE;
	xDiagCreateInfo.infoKind	:= asdiagCONFIGURED;
	xDiagCreateInfo();

	IF (xDiagCreateInfo.status = 0) THEN
		iIdent 		:= xDiagCreateInfo.ident;
		iNrEntries	:= xDiagCreateInfo.nrEntries;
	END_IF;

	(** 2.2: search names and get correct path of configured X20CS1030_xxx_xx_GCB module *)
	memset(ADR(sLabelInfo),	 	0, SIZEOF(sLabelInfo));
	FOR iIndex := 0 TO iNrEntries - 1 DO
		xDiagGetStrInfo.enable		:= TRUE;
		xDiagGetStrInfo.ident		:= iIdent;
		xDiagGetStrInfo.index		:= iIndex;
		xDiagGetStrInfo.infoCode	:= asdiagHARDWARE_MODULE_NAME;
		xDiagGetStrInfo.pBuffer		:= ADR(sLabelInfo);
		xDiagGetStrInfo.bufferLen	:= SIZEOF(sLabelInfo) - 1;
		xDiagGetStrInfo();

		IF xDiagGetStrInfo.status = 0 THEN
			IF FIND(sLabelInfo, 'X20CS1030') <> 0 THEN
				IF FIND(sLabelInfo, 'GCB') <> 0 THEN
					xDiagGetStrInfo.infoCode	:= asdiagPATH;
					xDiagGetStrInfo.pBuffer		:= ADR(sAddrInfo);
					xDiagGetStrInfo.bufferLen	:= SIZEOF(sAddrInfo) - 1;
					xDiagGetStrInfo();
					IF (xDiagGetStrInfo.status = 0) THEN
						sRTUAddr	:=	CONCAT(sAddrInfo,'.IF1');
					END_IF
					EXIT;
				END_IF
			END_IF
		END_IF
	END_FOR

	(** 2.3: free ressources of AsIODiag *)
	xDiagDisposeInfo.enable := TRUE;
	xDiagDisposeInfo.ident  := iIdent;
	xDiagDisposeInfo();

	(** 3: If no Address was found deactivate task and end init now *)
	IF sRTUAddr = '' THEN
		bDeactivate_Task := TRUE;
		RETURN;
	ELSE
		MM2VIS.tGCB[1].bEna	:=	TRUE;
	END_IF

	(** 4: Global initialization of master *)
	//Physical properties	/PHY	RS232|RS422|RS485| TTY|RS422BUS
	//Parity				/PA		N|E|O|H|L
	//Data bits				/DB		7|8
	//Stop bits				/SB		1|2
	//Baud rate				/BD		300-115200
	//possible to increase the amount of masters
	xMBDO_Master[0].bEnable				:=	TRUE;
	xMBDO_Master[0].pName_Module		:=	ADR('Synchronization');	//Name of this Module
	xMBDO_Master[0].pName_Task			:=	ADR('LV_GCB');			//Name of this Task
	xMBDO_Master[0].iMemType			:=	doUSRRAM;				//Memory where the Modbus data object should be created
	xMBDO_Master[0].pCmd				:=	ADR(tCmd[0]);			//Pointer to Master command structure
	xMBDO_Master[0].tCfg.sMode			:=	'/PHY=RS485 /PA=E /DB=8 /SB=1 /BD=19200'; //see above
	xMBDO_Master[0].tCfg.iTimeOut		:=	300;					//Timeout in ms (value must be a multiple of 10)
	xMBDO_Master[0].tCfg.bASCII			:=	FALSE;					//ModBus mode (0 = RTU / 1 = ASCII)
	xMBDO_Master[0].tCfg.iID			:=	1;						//ID of Master (Zero not accepted)
	xMBDO_Master[0].tSlave				:=	ADR(tSlave);			//Pointer to Slave structure
	tCmd[0].bOpen						:=	TRUE;					//open communication

	(** 5: Local initialization of masters *)
	(** 5.1: Local initialization of master #1 *)
	xMBDO_Master[0].tCfg.sDevice	:=	sRTUAddr;		//Address of X20CS1030
	xMBDO_Master[0].tCfg.sFile		:=	'CFG_GCB';		//Data object name

	(** 6: Local initialization of slaves*)
	//Master that is connected to this slave	iMaster
	//Slaves name								sName
	//Slaves address on ModBus					iAdr
	//Additional info e.g. cubicle number		iInfo

	(** 6.1: Slaves *)
	tSlave[0].iMaster	:=	1;
	tSlave[0].sName		:=	'ABB EMAX 2';
	tSlave[0].iAdr		:=	247;				//ABB: default
	tSlave[0].iInfo		:=	1;					//not needed at moment

	tSlave[1].iMaster	:=	1;
	tSlave[1].sName		:=	'Schneider MTZ';
	tSlave[1].iAdr		:=	17;					//SE: must be set on IFM
	tSlave[1].iInfo		:=	1;					//not needed at moment

	//Modbus Function Code					iFC
	//Modbus Register Length				iLen
	//Modbus Register Offset				iOffs
	//Word offset in extra Memory array		iWordOffs
	//Bit offset in extra Memory array		iBitOffs

	(** 6.2: Command lines for each slave *)

	tSlave[0].tLine[0].tDef.iFC				:=	4;
	tSlave[0].tLine[0].tDef.iLen			:=	4;
	tSlave[0].tLine[0].tDef.iOffs			:=	20;			//Contact wear

	tSlave[0].tLine[1].tDef.iFC				:=	4;
	tSlave[0].tLine[1].tDef.iLen			:=	1;
	tSlave[0].tLine[1].tDef.iOffs			:=	30;			//read programming failure codes

	tSlave[0].tLine[2].tDef.iFC				:=	4;
	tSlave[0].tLine[2].tDef.iLen			:=	6;
	tSlave[0].tLine[2].tDef.iOffs			:=	100;		//read Current measures

	tSlave[0].tLine[3].tDef.iFC				:=	4;
	tSlave[0].tLine[3].tDef.iLen			:=	3;
	tSlave[0].tLine[3].tDef.iOffs			:=	154;		//read Voltage measures

	tSlave[0].tLine[4].tDef.iFC				:=	4;
	tSlave[0].tLine[4].tDef.iLen			:=	1;
	tSlave[0].tLine[4].tDef.iOffs			:=	652;		//read Primary Voltage

	tSlave[0].tLine[6].tDef.iFC				:=	4;
	tSlave[0].tLine[6].tDef.iLen			:=	8;
	tSlave[0].tLine[6].tDef.iOffs			:=	700;		//read L (ANSI 49)

	tSlave[0].tLine[7].tDef.iFC				:=	4;
	tSlave[0].tLine[7].tDef.iLen			:=	9;
	tSlave[0].tLine[7].tDef.iOffs			:=	710;		//read S (ANSI 50TD, 68, 51N)

	tSlave[0].tLine[8].tDef.iFC				:=	4;
	tSlave[0].tLine[8].tDef.iLen			:=	4;
	tSlave[0].tLine[8].tDef.iOffs			:=	720;		//read I (ANSI 50)

	tSlave[0].tLine[9].tDef.iFC				:=	16;
	tSlave[0].tLine[9].tDef.iLen			:=	2;
	tSlave[0].tLine[9].tDef.iOffs			:=	711;		//write S (ANSI 50TD, 68, 51N)

	tSlave[0].tLine[10].tDef.iFC			:=	6;
	tSlave[0].tLine[10].tDef.iLen			:=	1;
	tSlave[0].tLine[10].tDef.iOffs			:=	721;		//write I (ANSI 50)

	tSlave[0].tLine[11].tDef.iFC			:=	4;
	tSlave[0].tLine[11].tDef.iLen			:=	1;
	tSlave[0].tLine[11].tDef.iOffs			:=	40;			//read Information

	tSlave[0].tLine[12].tDef.iFC			:=	4;
	tSlave[0].tLine[12].tDef.iLen			:=	1;
	tSlave[0].tLine[12].tDef.iOffs			:=	504;		//read Nom Current

	tSlave[0].tLine[13].tDef.iFC			:=	16;
	tSlave[0].tLine[13].tDef.iLen			:=	2;
	tSlave[0].tLine[13].tDef.iOffs			:=	0;			//write Commands

	tSlave[0].tLine[14].tDef.iFC			:=	16;
	tSlave[0].tLine[14].tDef.iLen			:=	2;
	tSlave[0].tLine[14].tDef.iOffs			:=	701;		//write L (ANSI 49)

	//Schneider MTZ:
	tSlave[1].tLine[0].tDef.iFC				:=	4;
	tSlave[1].tLine[0].tDef.iLen			:=	4;
	tSlave[1].tLine[0].tDef.iOffs			:=	35204-1;	//Op cnt + Trip counter in uint32

	tSlave[1].tLine[1].tDef.iFC				:=	4;
	tSlave[1].tLine[1].tDef.iLen			:=	2;
	tSlave[1].tLine[1].tDef.iOffs			:=	32000-1;	//0 = closed, 1= tripped

	tSlave[1].tLine[2].tDef.iFC				:=	4;
	tSlave[1].tLine[2].tDef.iLen			:=	6;
	tSlave[1].tLine[2].tDef.iOffs			:=	32028-1;	//real time current L1-L3 float 32bit

	tSlave[1].tLine[3].tDef.iFC				:=	4;
	tSlave[1].tLine[3].tDef.iLen			:=	2;
	tSlave[1].tLine[3].tDef.iOffs			:=	21013-1;	//real time avg voltage float 32bit

	tSlave[1].tLine[4].tDef.iFC				:=	4;
	tSlave[1].tLine[4].tDef.iLen			:=	4;
	tSlave[1].tLine[4].tDef.iOffs			:=	8153-1;		//nom voltage and current in 32bit float

	tSlave[1].tLine[5].tDef.iFC				:=	4;
	tSlave[1].tLine[5].tDef.iLen			:=	2;
	tSlave[1].tLine[5].tDef.iOffs			:=	24001-1;	//contact wear in 32bit float

	tSlave[1].tLine[6].tDef.iFC				:=	4;
	tSlave[1].tLine[6].tDef.iLen			:=	4;
	tSlave[1].tLine[6].tDef.iOffs			:=	45025-1;	//long time overcurrent in 32bit float

	tSlave[1].tLine[7].tDef.iFC				:=	4;
	tSlave[1].tLine[7].tDef.iLen			:=	4;
	tSlave[1].tLine[7].tDef.iOffs			:=	45035-1;	//short time overcurrent in 32bit float

	tSlave[1].tLine[8].tDef.iFC				:=	4;
	tSlave[1].tLine[8].tDef.iLen			:=	3;
	tSlave[1].tLine[8].tDef.iOffs			:=	45044-1;	//instantaneous overcurrent in 32bit float

	tSlave[1].tLine[9].tDef.iFC				:=	4;
	tSlave[1].tLine[9].tDef.iLen			:=	1;
	tSlave[1].tLine[9].tDef.iOffs			:=	15330-1;	// TBD

	tSlave[1].tLine[10].tDef.iFC			:=	16;
	tSlave[1].tLine[10].tDef.iLen			:=	14;
	tSlave[1].tLine[10].tDef.iOffs			:=	8000-1;			//write Commands

	tSlave[1].tLine[11].tDef.iFC			:=	4;
	tSlave[1].tLine[11].tDef.iLen			:=	5;
	tSlave[1].tLine[11].tDef.iOffs			:=	8020-1;			//check write Commands

	(** 7: check complete configuration *)
	bError_Conf	:=	MSC_MB_DataCheck(ADR(tSlave)) > 0;

	(** 8: Special modbus commands for Schneider *)
	//	User profile Default password
	//	Administrator ‘0000’ = 0x30303030 => 12336 & 12336
	//	Services ‘1111’ = 0x31313131
	//	Engineer ‘2222’ = 0x32323232
	//	Operator ‘3333’ = 0x33333333

	(** 8.1: Open Setup Session *)
	tIF_Session_Open.bExec		:=	TRUE;
	tIF_Session_Open.iData[0]	:=	1930;
	tIF_Session_Open.iData[1]	:=	10;
	tIF_Session_Open.iData[2]	:=	5377;
	tIF_Session_Open.iData[3]	:=	1;
	tIF_Session_Open.iData[4]	:=	12336;
	tIF_Session_Open.iData[5]	:=	12336;

	(** 8.2: Close Setup Session *)
	tIF_Session_Close.bExec		:=	TRUE;
	tIF_Session_Close.iData[0]	:=	1933;
	tIF_Session_Close.iData[1]	:=	14;
	tIF_Session_Close.iData[2]	:=	5377;
	tIF_Session_Close.iData[3]	:=	1;
	tIF_Session_Close.iData[4]	:=	12336;
	tIF_Session_Close.iData[5]	:=	12336;

	(** 8.3: Apply Settings *)
	tIF_Session_Apply.bExec		:=	TRUE;
	tIF_Session_Apply.iData[0]	:=	1932;
	tIF_Session_Apply.iData[1]	:=	14;
	tIF_Session_Apply.iData[2]	:=	5377;
	tIF_Session_Apply.iData[3]	:=	1;
	tIF_Session_Apply.iData[4]	:=	12336;
	tIF_Session_Apply.iData[5]	:=	12336;

	(** 8.4: Submit Long Time Over Current Protection Settings *)
	tIF_Session_Change1.bExec		:=	TRUE;
	tIF_Session_Change1.iData[0]	:=	51593;
	tIF_Session_Change1.iData[1]	:=	26;
	tIF_Session_Change1.iData[2]	:=	5377;
	tIF_Session_Change1.iData[3]	:=	1;
	tIF_Session_Change1.iData[4]	:=	12336;
	tIF_Session_Change1.iData[5]	:=	12336;
	// 6&7: SessionKey
	tIF_Session_Change1.iData[8]	:=	1;		// Group A = 1
	tIF_Session_Change1.iData[9]	:=	65535;	// Reserved
	// 10&11: Range - / Step 0.1A
	// 12&13: Range 0.5 - 24.0 / Step 0.5s

	(** 8.5: Submit Short Time Over Current Protection Settings *)
	tIF_Session_Change2.bExec		:=	TRUE;
	tIF_Session_Change2.iData[0]	:=	51594;
	tIF_Session_Change2.iData[1]	:=	26;
	tIF_Session_Change2.iData[2]	:=	5377;
	tIF_Session_Change2.iData[3]	:=	1;
	tIF_Session_Change2.iData[4]	:=	12336;
	tIF_Session_Change2.iData[5]	:=	12336;
	// 6&7: SessionKey
	tIF_Session_Change2.iData[8]	:=	1;	// Group A = 1
	tIF_Session_Change2.iData[9]	:=	0;	// I²t = On, 0: I²t = Off
	// 10&11: Range 1.5 - 10.0 / Step 0.1
	// 12&13: Range 0.0 - 0.4 / Step 0.1s

	(** 8.6: Submit Instantaneous Protection Settings *)
	tIF_Session_Change3.bExec		:=	TRUE;
	tIF_Session_Change3.iData[0]	:=	51595;
	tIF_Session_Change3.iData[1]	:=	22;
	tIF_Session_Change3.iData[2]	:=	5377;
	tIF_Session_Change3.iData[3]	:=	1;
	tIF_Session_Change3.iData[4]	:=	12336;
	tIF_Session_Change3.iData[5]	:=	12336;
	// 6&7: SessionKey
	tIF_Session_Change3.iData[8]	:=	16#0101;	//MSB: 1 = On	// LSB: Group A = 1
	// 9&10: Range 2.0 - 15.0 / Step 0.1
	tIF_Session_Change3.iData[11]	:=	1;	//  0 = Standart, 1 = Fast

	(** 9: Special modbus commands for ABB *)
	(** 9.1: ABB Command open program session *)
	tIF_ABB_Open.bExec		:=	TRUE;
	tIF_ABB_Open.iData[0]	:=	4;
	tIF_ABB_Open.iData[1]	:=	0;

	(** 9.2: ABB Command close program session	*)
	tIF_ABB_Close.bExec		:=	TRUE;
	tIF_ABB_Close.iData[0]	:=	6;
	tIF_ABB_Close.iData[1]	:=	0;

END_PROGRAM
```

#### LV_GCB.var
```iecst
VAR
	xWAIT : {REDUND_UNREPLICABLE} WAIT_CYCLIC := (0); (*Timer for LV GCB state machine*)
	xTIMEOUT : {REDUND_UNREPLICABLE} WAIT_CYCLIC := (0); (*Timeout timer for LV GCB state machine*)
	i : {REDUND_UNREPLICABLE} USINT; (*Counter*)
	iSessionKey1 : {REDUND_UNREPLICABLE} UINT := 0; (*Schneider command session Key #1*)
	iSessionKey0 : {REDUND_UNREPLICABLE} UINT := 0; (*Schneider command session Key #0*)
	iIndex : {REDUND_UNREPLICABLE} UDINT; (*Index of actual read module*)
	iIdent : {REDUND_UNREPLICABLE} UDINT; (*Ident from xDiagCreateInfo*)
	iNrEntries : {REDUND_UNREPLICABLE} UDINT; (*Number of configured modules from xDiagCreateInfo*)
	xTON_ParaSetup_Ok : {REDUND_UNREPLICABLE} TON := (0); (*Time delay for Parameter setup okay*)
	xTON_Rel_MBMaster : {REDUND_UNREPLICABLE} TON := (0); (*Time delay for ModBus master FUB*)
	xTOF_ParaSaved_5s : {REDUND_UNREPLICABLE} TOF := (0); (*Time delay for Parameters saved operating message*)
	tiRel_MBMaster : {REDUND_UNREPLICABLE} TIME := T#1S; (*Time delay for ModBus master FUB*)
	tiParaSetup_Ok : {REDUND_UNREPLICABLE} TIME := T#10S; (*Time delay for Parameter setup okay*)
	sLabelInfo : {REDUND_UNREPLICABLE} STRING[50]; (*Includes label of configured module*)
	sRTUAddr : {REDUND_UNREPLICABLE} STRING[50]; (*Modbus RTU IF PLC address string*)
	sAddrInfo : {REDUND_UNREPLICABLE} STRING[50]; (*Includes address of configured modul*)
	rFactors : {REDUND_UNREPLICABLE} REAL := 0.0; (*Factors that are selectable for over current protection*)
	rFactor_Isd : {REDUND_UNREPLICABLE} REAL := 0.0; (*Schneider delayed over current protection factor*)
	rFactor_Ii : {REDUND_UNREPLICABLE} REAL := 0.0; (*Schneider instantaneous over current protection factor*)
	rTemp : {REDUND_UNREPLICABLE} REAL := 0.0; (*Schneider temporary calculation variable*)
	xMBDO_Master : {REDUND_UNREPLICABLE} ARRAY[0.._MB_DEVICES_MAX] OF MSC_MBDOMaster; (*Modbus master FUB*)
	tSlave : {REDUND_UNREPLICABLE} ARRAY[0.._MB_SLAVES_MAX] OF MB_Reg_Slaves; (*Modbus slave structure*)
	tIF_Session_Change1 : {REDUND_UNREPLICABLE} MB_Reg_Interface := (0); (*Predefined ModBus command*)
	tIF_Session_Open : {REDUND_UNREPLICABLE} MB_Reg_Interface := (0); (*Predefined ModBus command*)
	tIF_Session_Apply : {REDUND_UNREPLICABLE} MB_Reg_Interface := (0); (*Predefined ModBus command*)
	tIF_Session_Close : {REDUND_UNREPLICABLE} MB_Reg_Interface := (0); (*Predefined ModBus command*)
	tIF_Session_Change2 : {REDUND_UNREPLICABLE} MB_Reg_Interface := (0); (*Predefined ModBus command*)
	tIF_Session_Change3 : {REDUND_UNREPLICABLE} MB_Reg_Interface := (0); (*Predefined ModBus command*)
	tIF_ABB_Close : {REDUND_UNREPLICABLE} MB_Reg_Interface := (0); (*Predefined ModBus command*)
	tIF_ABB_Open : {REDUND_UNREPLICABLE} MB_Reg_Interface := (0); (*Predefined ModBus command*)
	tCmd : {REDUND_UNREPLICABLE} ARRAY[0.._MB_DEVICES_MAX] OF MB_Commands; (*ModBus master FUB command structure*)
	eState_GCB : {REDUND_UNREPLICABLE} LV_GCB := _GCB_INIT; (*Current LV GCB State*)
	eState_GCB_Old : {REDUND_UNREPLICABLE} LV_GCB := _GCB_INIT; (*Old LV GCB State*)
	eState_GCB_TO : {REDUND_UNREPLICABLE} LV_GCB := _GCB_INIT; (*Timeout LV GCB State*)
	iType_Old : {REDUND_UNREPLICABLE} INT := 0; (*Old GCB Type (1=ABB, 2=Schneider)*)
	xDiagGetStrInfo : {REDUND_UNREPLICABLE} DiagGetStrInfo; (*Get name of configured modules*)
	xDiagDisposeInfo : {REDUND_UNREPLICABLE} DiagDisposeInfo; (*Free ressources of AsIODiag*)
	xDiagCreateInfo : {REDUND_UNREPLICABLE} DiagCreateInfo; (*Get number of configured modules*)
	bError_Conf : {REDUND_UNREPLICABLE} BOOL := 0; (*Error in Slave configuration*)
	bInit : {REDUND_UNREPLICABLE} BOOL := 0; (*Init Bit in LV GCB state machine*)
	bABB : {REDUND_UNREPLICABLE} BOOL := 0; (*ABB = Current GCB Type*)
	bSE : {REDUND_UNREPLICABLE} BOOL := 0; (*Schneider = Current GCB Type*)
	bDeactivate_Task : {REDUND_UNREPLICABLE} BOOL := 0; (*Deactivates whole Task*)
	bClear : {REDUND_UNREPLICABLE} BOOL := 0; (*Clears displayed data on HMI*)
	bABB_Remote : {REDUND_UNREPLICABLE} BOOL := 0; (*Checks if ABB LV GCB is in remote mode*)
END_VAR
```

#### MSC_MB.fun - Exported functions and function blocks
```iecst
(********************************************************************
 * COPYRIGHT -- INNIO, MSC
 ********************************************************************
 * Library: MSC_MB
 * File: MSC_MB.fun
 * Author: Hohensinner Michael
 * Created: April 29, 2021
 ********************************************************************
 * Functions and function blocks of library MSC_MB
 ********************************************************************)
(* ModBus Master function block 4 easy use *)

{REDUND_OK} {REDUND_UNREPLICABLE} FUNCTION_BLOCK MSC_MBMaster
	VAR_INPUT
		bEnable : {REDUND_UNREPLICABLE} BOOL;
		tCfg : {REDUND_UNREPLICABLE} MBM_Config;
		tCmd : REFERENCE TO MB_Commands;
	END_VAR
	VAR_OUTPUT
		eState : {REDUND_UNREPLICABLE} MB_State_Enum;
		eError : {REDUND_UNREPLICABLE} MB_State_Enum;
		iError : {REDUND_UNREPLICABLE} UINT;
		bExec : {REDUND_UNREPLICABLE} BOOL;
		iRecNum : {REDUND_UNREPLICABLE} UINT;
		iStatus : {REDUND_UNREPLICABLE} UINT;
	END_VAR
	VAR
		xMBMOpen : {REDUND_UNREPLICABLE} MBMOpen;
		xMBMaster : {REDUND_UNREPLICABLE} MBMaster;
		xMBMClose : {REDUND_UNREPLICABLE} MBMClose;
	END_VAR
END_FUNCTION_BLOCK
(* ModBus Slave function block 4 easy use *)

{REDUND_OK} {REDUND_UNREPLICABLE} FUNCTION_BLOCK MSC_MBSlave
	VAR_INPUT
		bEnable : {REDUND_UNREPLICABLE} BOOL;
		tCfg : {REDUND_UNREPLICABLE} MBS_Config;
		tCmd : REFERENCE TO MB_Commands;
	END_VAR
	VAR_OUTPUT
		eState : {REDUND_UNREPLICABLE} MB_State_Enum;
		eError : {REDUND_UNREPLICABLE} MB_State_Enum;
		iError : {REDUND_UNREPLICABLE} UINT;
	END_VAR
	VAR
		xMBSOpen : {REDUND_UNREPLICABLE} MBSOpen;
		xMBSlave : {REDUND_UNREPLICABLE} MBSlave;
		xMBSClose : {REDUND_UNREPLICABLE} MBSClose;
	END_VAR
END_FUNCTION_BLOCK

{REDUND_OK} {REDUND_UNREPLICABLE} FUNCTION_BLOCK MSC_MB_DataLine
	VAR_INPUT
		pName_Module : {REDUND_UNREPLICABLE} UDINT;
		pName_Task : {REDUND_UNREPLICABLE} UDINT;
		pName_Struct : {REDUND_UNREPLICABLE} UDINT;
		iIdx_Slave : {REDUND_UNREPLICABLE} USINT;
		iIdx_Line : {REDUND_UNREPLICABLE} USINT;
		iFC : {REDUND_UNREPLICABLE} USINT;
		iAdr_Slave : {REDUND_UNREPLICABLE} USINT;
		iOffset : {REDUND_UNREPLICABLE} UINT;
		iLength : {REDUND_UNREPLICABLE} UINT;
	END_VAR
	VAR_OUTPUT
		iData : {REDUND_UNREPLICABLE} ARRAY[0.._MB_DATALINE_MAX] OF USINT;
		iStrLen : {REDUND_UNREPLICABLE} UDINT;
		bError : {REDUND_UNREPLICABLE} BOOL;
	END_VAR
	VAR
		sTemp : {REDUND_UNREPLICABLE} STRING[7];
		sData : {REDUND_UNREPLICABLE} STRING[_MB_DATALINE_MAX];
		iBegin : {REDUND_UNREPLICABLE} UDINT;
	END_VAR
END_FUNCTION_BLOCK

{REDUND_OK} {REDUND_UNREPLICABLE} FUNCTION_BLOCK MSC_MB_DataSet
	VAR_INPUT
		pName_Module : {REDUND_UNREPLICABLE} UDINT;
		pName_Task : {REDUND_UNREPLICABLE} UDINT;
		pName_Struct : {REDUND_UNREPLICABLE} UDINT;
		iIdx_Slave : {REDUND_UNREPLICABLE} USINT;
		iAdr_Slave : {REDUND_UNREPLICABLE} USINT;
		tLine : {REDUND_UNREPLICABLE} ARRAY[0.._MB_CMD_MAX] OF MB_Reg_Line;
	END_VAR
	VAR_OUTPUT
		iData : {REDUND_UNREPLICABLE} ARRAY[0.._MB_DATASET_MAX] OF USINT;
		iStrLen : {REDUND_UNREPLICABLE} UDINT;
		bEmpty : {REDUND_UNREPLICABLE} BOOL;
		bError : {REDUND_UNREPLICABLE} BOOL;
	END_VAR
	VAR
		i : {REDUND_UNREPLICABLE} UDINT;
		xLine : {REDUND_UNREPLICABLE} MSC_MB_DataLine;
	END_VAR
END_FUNCTION_BLOCK

{REDUND_OK} {REDUND_UNREPLICABLE} FUNCTION_BLOCK MSC_MB_DOCreate
	VAR_INPUT
		bEnable : {REDUND_UNREPLICABLE} BOOL;
		pName : {REDUND_UNREPLICABLE} UDINT;
		pCpyData : {REDUND_UNREPLICABLE} UDINT;
		iMemType : {REDUND_UNREPLICABLE} USINT;
		iLen : {REDUND_UNREPLICABLE} UDINT;
	END_VAR
	VAR_OUTPUT
		eState : {REDUND_UNREPLICABLE} MB_State_Enum;
		bDone : {REDUND_UNREPLICABLE} BOOL;
	END_VAR
	VAR
		xDatObjInfo : {REDUND_UNREPLICABLE} DatObjInfo;
		xDatObjDelete : {REDUND_UNREPLICABLE} DatObjDelete;
		xDatObjCreate : {REDUND_UNREPLICABLE} DatObjCreate;
	END_VAR
END_FUNCTION_BLOCK

{REDUND_OK} {REDUND_UNREPLICABLE} FUNCTION_BLOCK MSC_MBDOMaster
	VAR_INPUT
		bEnable : {REDUND_UNREPLICABLE} BOOL; (*Enables the start of the communication, block will configure itself even without enable bit*)
		pName_Module : {REDUND_UNREPLICABLE} UDINT; (*pointer to name of application module, set to zero if no module is used*)
		pName_Task : {REDUND_UNREPLICABLE} UDINT; (*pointer to name of task, set to zero if variable is global*)
		pName_Struct : {REDUND_UNREPLICABLE} UDINT; (*pointer to name of variable, set to zero if default name 'tSlave' is used*)
		pCmd : {REDUND_UNREPLICABLE} UDINT; (*pointer to command structure*)
		tCfg : {REDUND_UNREPLICABLE} MBM_Config; (*Configuration of master*)
		tSlave : REFERENCE TO ARRAY[0.._MB_SLAVES_MAX] OF MB_Reg_Slaves; (*Configuration of all connected slaves*)
		iMemType : {REDUND_UNREPLICABLE} USINT; (*Target memory in which the data object is to be saved,  e.g. doTEMP, doUSRRAM, doUSRROM, ...*)
	END_VAR
	VAR_OUTPUT
		eError : {REDUND_UNREPLICABLE} MB_State_Enum;
		eState : {REDUND_UNREPLICABLE} MB_State_Enum;
		bExec : {REDUND_UNREPLICABLE} BOOL;
		iRecNum : {REDUND_UNREPLICABLE} UINT;
		iLog : {REDUND_UNREPLICABLE} ARRAY[0.._MB_SLAVES_MAX] OF UINT;
		iStatus : {REDUND_UNREPLICABLE} UINT;
		bError : {REDUND_UNREPLICABLE} BOOL;
	END_VAR
	VAR
		xMB_DOCreate : {REDUND_UNREPLICABLE} MSC_MB_DOCreate;
		xMB_DataSet : {REDUND_UNREPLICABLE} MSC_MB_DataSet;
		xMB_Master : {REDUND_UNREPLICABLE} MSC_MBMaster;
		xTON_Reset_Log : {REDUND_UNREPLICABLE} ARRAY[0.._MB_SLAVES_MAX] OF TON;
		iData : {REDUND_UNREPLICABLE} ARRAY[0.._MB_DATAOBJ_MAX] OF USINT;
		iLen : {REDUND_UNREPLICABLE} UDINT;
		iEntry : {REDUND_UNREPLICABLE} USINT;
		j : {REDUND_UNREPLICABLE} INT;
		i : {REDUND_UNREPLICABLE} INT;
		iRecNum_Old : {REDUND_UNREPLICABLE} UINT;
		iListSlave : {REDUND_UNREPLICABLE} ARRAY[0.._MB_ENTRIES_MAX] OF USINT;
		iListCmd : {REDUND_UNREPLICABLE} ARRAY[0.._MB_ENTRIES_MAX] OF USINT;
	END_VAR
END_FUNCTION_BLOCK

{REDUND_OK} FUNCTION MSC_MB_DataCheck : UINT
	VAR_INPUT
		tSlave : REFERENCE TO ARRAY[0.._MB_SLAVES_MAX] OF MB_Reg_Slaves; (*Configuration of all connected slaves*)
	END_VAR
	VAR
		j : USINT;
		i : USINT;
	END_VAR
END_FUNCTION

{REDUND_OK} FUNCTION MSC_MB_RegUpdate : USINT
	VAR_INPUT
		tSlave : REFERENCE TO MB_Reg_Slaves;
		iError : REFERENCE TO UINT;
		iRead : REFERENCE TO UINT;
		iWrite : REFERENCE TO UINT;
		bEnaRead : BOOL;
		bEnaWrite : BOOL;
	END_VAR
	VAR
		iByteSize : UDINT;
		i : UINT;
		x : USINT;
		iTemp : ARRAY[0.._MB_DATA_ARRAY_MAX] OF UINT;
		bError : BOOL;
	END_VAR
END_FUNCTION

{REDUND_OK} FUNCTION UINT_TWO_REAL : REAL
	VAR_INPUT
		IN1 : UINT;
		IN2 : UINT;
	END_VAR
END_FUNCTION

{REDUND_OK} FUNCTION UINT_TWO_UDINT : UDINT
	VAR_INPUT
		IN1 : UINT;
		IN2 : UINT;
	END_VAR
END_FUNCTION

{REDUND_OK} FUNCTION STEP : REAL
	VAR_INPUT
		IN : REAL;
		STEPSIZE : REAL;
	END_VAR
END_FUNCTION

{REDUND_OK} FUNCTION_BLOCK WAIT_CYCLIC
	VAR_INPUT
		IN : {REDUND_UNREPLICABLE} UINT;
	END_VAR
	VAR_OUTPUT
		Q : {REDUND_UNREPLICABLE} BOOL;
	END_VAR
	VAR
		CNT : UINT;
	END_VAR
END_FUNCTION_BLOCK

FUNCTION SET_BIT_UINT_ARRAY : BOOL
	VAR_INPUT
		bSet : BOOL;
		iBit : UINT;
		iArray : REFERENCE TO ARRAY[0.._MB_DATA_ARRAY_MAX] OF UINT;
	END_VAR
END_FUNCTION

FUNCTION GET_BIT_UINT_ARRAY : BOOL
	VAR_INPUT
		iBit : UINT;
		iArray : REFERENCE TO ARRAY[0.._MB_DATA_ARRAY_MAX] OF UINT;
	END_VAR
END_FUNCTION
```
